	16#000005B8:
		F_EtherCAT_VendorIDtoString := 'Tarasheh System Pishro (tsPishro) Co., Ltd.';

	16#000005B9:
		F_EtherCAT_VendorIDtoString := 'CS-Lab s.c. Janusz Wawak, Andrzej Rogozynski, Szymon Paprocki';

	16#000005BA:
		F_EtherCAT_VendorIDtoString := 'Elitron IPM s.r.l.';

	16#000005BB:
		F_EtherCAT_VendorIDtoString := 'KORYO ELECTRONICS CO.,LTD.';

	16#000005BC:
		F_EtherCAT_VendorIDtoString := 'Shihlin Electric & Engineering Corporation';

	16#000005BD:
		F_EtherCAT_VendorIDtoString := 'Kookmin University, Graduate School of Automotive Engineering';

	16#000005BE:
		F_EtherCAT_VendorIDtoString := 'Techmation Co., Ltd.';

	16#000005BF:
		F_EtherCAT_VendorIDtoString := 'ZAPI S.p.A.';

	16#000005C0:
		F_EtherCAT_VendorIDtoString := 'Claus Pribbernow Mikrosystementwicklung eProcessorSolutions';

	16#000005C1:
		F_EtherCAT_VendorIDtoString := 'Pragati Automation Pvt. Ltd.';

	16#000005C2:
		F_EtherCAT_VendorIDtoString := 'Siemens Industry Software B.V.';

	16#000005C3:
		F_EtherCAT_VendorIDtoString := 'MicroNova AG';

	16#000005C4:
		F_EtherCAT_VendorIDtoString := 'XiAn Aerospace Precision Electromechanical Institute';

	16#000005C5:
		F_EtherCAT_VendorIDtoString := 'Dr. Mergenthaler GmbH & Co. KG';

	16#000005C6:
		F_EtherCAT_VendorIDtoString := 'China National Machinery Industry Corporation';

	16#000005C7:
		F_EtherCAT_VendorIDtoString := 'Berufliches Schulzentrum Hof, Staatliche Fachschule fur Technik';

	16#000005C8:
		F_EtherCAT_VendorIDtoString := 'NDR Co., Ltd';

	16#000005C9:
		F_EtherCAT_VendorIDtoString := '"NPK MSA" LLC';

	16#000005CA:
		F_EtherCAT_VendorIDtoString := 'Southeast University, School of Mechanical Engineering';

	16#000005CB:
		F_EtherCAT_VendorIDtoString := 'Shanghai Baosight Software Co., Ltd.';

	16#000005CC:
		F_EtherCAT_VendorIDtoString := 'Hakko Electronics Co., Ltd.';

	16#000005CD:
		F_EtherCAT_VendorIDtoString := 'GMK electronic design GmbH';

	16#000005CE:
		F_EtherCAT_VendorIDtoString := 'SIMTEC Elektronik GmbH';

	16#000005D0:
		F_EtherCAT_VendorIDtoString := 'TEConcept GmbH';

	16#000005D1:
		F_EtherCAT_VendorIDtoString := 'ESS Co., Ltd.';

	16#000005D3:
		F_EtherCAT_VendorIDtoString := 'MABI AG - Robotic';

	16#000005D4:
		F_EtherCAT_VendorIDtoString := 'OnRobot Hungary Kft';

	16#000005D5:
		F_EtherCAT_VendorIDtoString := 'TMEIC Corporation';

	16#000005D6:
		F_EtherCAT_VendorIDtoString := 'WITTENSTEIN ternary Co.,Ltd.';

	16#000005D7:
		F_EtherCAT_VendorIDtoString := 'Shanghai Friendess Electronic Technology Co., Ltd.';

	16#000005D8:
		F_EtherCAT_VendorIDtoString := 'Aversan Inc.';

	16#000005DA:
		F_EtherCAT_VendorIDtoString := 'Lorch Schweitechnik GmbH';

	16#000005D9:
		F_EtherCAT_VendorIDtoString := 'LOTES (GuangZhou) CO., LTD.';

	16#000005DB:
		F_EtherCAT_VendorIDtoString := 'Sungkyunkwan University, School of Mechanical Engineering';

	16#000005DC:
		F_EtherCAT_VendorIDtoString := 'Tsinghua University, Graduate School at Shenzhen';

	16#000005DD:
		F_EtherCAT_VendorIDtoString := 'Universidad de los Andes, Faculty of Engineering';

	16#000005DE:
		F_EtherCAT_VendorIDtoString := 'PFU LIMITED';

	16#000005DF:
		F_EtherCAT_VendorIDtoString := 'Slovak University of Technology in Bratislava, Faculty of Electrical Engineering and Information Technology';

	16#000005E0:
		F_EtherCAT_VendorIDtoString := 'Esomatec GmbH';

	16#000005E1:
		F_EtherCAT_VendorIDtoString := 'LS ELECTRIC Co., Ltd.';

	16#000005E2:
		F_EtherCAT_VendorIDtoString := 'StateCore B.V.';

	16#000005E3:
		F_EtherCAT_VendorIDtoString := 'KJ-Infinity Enterprises Inc.';

	16#000005E4:
		F_EtherCAT_VendorIDtoString := 'Center of Human-centered Interaction for Coexistence (CHIC)';

	16#000005E5:
		F_EtherCAT_VendorIDtoString := 'Littelfuse Selco A/S';

	16#000005E6:
		F_EtherCAT_VendorIDtoString := 'ITR GmbH Informationstechnologie Rauch';

	16#000005E8:
		F_EtherCAT_VendorIDtoString := 'University of Massachusetts at Amherst, Computer Science Department, Laboratory for Perceptual Robotics';

	16#000005E9:
		F_EtherCAT_VendorIDtoString := 'Pfeiffer Vacuum SAS';

	16#000005EA:
		F_EtherCAT_VendorIDtoString := 'AXOR INDUSTRIES s.n.c.';

	16#000005EB:
		F_EtherCAT_VendorIDtoString := 'QuadRep Electronics (Taiwan) Ltd.';

	16#000005EC:
		F_EtherCAT_VendorIDtoString := 'Herrmann Ultraschalltechnik GmbH & Co. KG';

	16#000005ED:
		F_EtherCAT_VendorIDtoString := 'Precizika Metrology, UAB';

	16#000005EE:
		F_EtherCAT_VendorIDtoString := 'Shanghai ReCAT Automation Control Technology Co., Ltd.';

	16#000005EF:
		F_EtherCAT_VendorIDtoString := 'U&R GmbH Hardware- und Systemdesign';

	16#000005F0:
		F_EtherCAT_VendorIDtoString := 'XiaMen MicroControl Technology Co., Ltd.';

	16#000005F1:
		F_EtherCAT_VendorIDtoString := 'The Oilgear Company';

	16#000005F2:
		F_EtherCAT_VendorIDtoString := 'MIE ELECTRONICS CO.,LTD. iSPC';

	16#000005F3:
		F_EtherCAT_VendorIDtoString := 'in-tech GmbH';

	16#000005F5:
		F_EtherCAT_VendorIDtoString := 'Starflight Electronics';

	16#000005F6:
		F_EtherCAT_VendorIDtoString := 'ZIEHL-ABEGG SE';

	16#000005F7:
		F_EtherCAT_VendorIDtoString := 'Ackermann Automation GmbH';

	16#000005F8:
		F_EtherCAT_VendorIDtoString := 'Helios Technologies, Inc.';

	16#000005F9:
		F_EtherCAT_VendorIDtoString := 'Italsensor s.r.l.';

	16#000005FA:
		F_EtherCAT_VendorIDtoString := 'Minebea Intec Aachen GmbH & Co. KG';

	16#000005FB:
		F_EtherCAT_VendorIDtoString := 'Evergrid Solutions & Systems';

	16#000005FC:
		F_EtherCAT_VendorIDtoString := 'Germanjet Company Limited';

	16#000005FD:
		F_EtherCAT_VendorIDtoString := 'Mapacode Inc.';

	16#000005FE:
		F_EtherCAT_VendorIDtoString := 'BIBA - Bremer Institut fur Produktion und Logistik GmbH';

	16#000005FF:
		F_EtherCAT_VendorIDtoString := 'The University of Texas at Austin';

	16#00000600:
		F_EtherCAT_VendorIDtoString := 'OKI Nextech Co.,Ltd.';

	16#00000601:
		F_EtherCAT_VendorIDtoString := 'Condalo GmbH';

	16#00000602:
		F_EtherCAT_VendorIDtoString := 'Brooks Instrument, LLC';

	16#00000603:
		F_EtherCAT_VendorIDtoString := 'FLORIDA INSTITUTE FOR HUMAN & MACHINE COGNITION';

	16#00000604:
		F_EtherCAT_VendorIDtoString := 'Leica Geosystems AG';

	16#00000605:
		F_EtherCAT_VendorIDtoString := 'Nabtesco Corporation';

	16#00000606:
		F_EtherCAT_VendorIDtoString := 'BP&M Representacoes e Consultoria LTDA';

	16#00000607:
		F_EtherCAT_VendorIDtoString := 'MICRO-EPSILON Optronic GmbH';

	16#00000608:
		F_EtherCAT_VendorIDtoString := 'Diamond Technologies, Inc.';

	16#0000060A:
		F_EtherCAT_VendorIDtoString := 'ESTUN AUTOMATION CO.,LTD';

	16#0000060B:
		F_EtherCAT_VendorIDtoString := 'IMS Messsysteme GmbH';

	16#0000060C:
		F_EtherCAT_VendorIDtoString := 'MG Co., Ltd.';

	16#0000060D:
		F_EtherCAT_VendorIDtoString := 'Ferrotec (USA) Corporation - Temescal Division';

	16#0000060E:
		F_EtherCAT_VendorIDtoString := 'SICK IVP AB';

	16#0000060F:
		F_EtherCAT_VendorIDtoString := 'Oregon State University, School of Mechanical, Industrial and Manufacturing Engineering';

	16#00000610:
		F_EtherCAT_VendorIDtoString := 'SINFONIA TECHNOLOGY CO., LTD.';

	16#00000611:
		F_EtherCAT_VendorIDtoString := 'Pfeiffer Vacuum GmbH';

	16#00000612:
		F_EtherCAT_VendorIDtoString := 'Froude Hofmann Limited';

	16#00000613:
		F_EtherCAT_VendorIDtoString := 'SABO Elektronik GmbH';

	16#00000615:
		F_EtherCAT_VendorIDtoString := 'Bystronic Laser AG';

	16#00000616:
		F_EtherCAT_VendorIDtoString := 'Shanghai Kinway Technologies, Inc.';

	16#00000617:
		F_EtherCAT_VendorIDtoString := 'Avnet K.K.';

	16#00000618:
		F_EtherCAT_VendorIDtoString := 'LumaSense Technologies GmbH';

	16#00000619:
		F_EtherCAT_VendorIDtoString := 'BBH Products GmbH';

	16#0000061A:
		F_EtherCAT_VendorIDtoString := 'Hecht Automatisierungs-Systeme GmbH';

	16#0000061B:
		F_EtherCAT_VendorIDtoString := 'Xelmo AB';

	16#0000061C:
		F_EtherCAT_VendorIDtoString := 'Carl Zeiss Industrielle Messtechnik GmbH';

	16#0000061D:
		F_EtherCAT_VendorIDtoString := 'University of Genova, Faculty of Engineering';

	16#0000061E:
		F_EtherCAT_VendorIDtoString := 'JOT Automation Oy';

	16#0000061F:
		F_EtherCAT_VendorIDtoString := 'Sankyo Seisakusho Co.';

	16#00000620:
		F_EtherCAT_VendorIDtoString := 'ATV-Elektronik Ges.m.b.H.';

	16#00000621:
		F_EtherCAT_VendorIDtoString := 'Panasonic Industry Co., Ltd.';

	16#00000622:
		F_EtherCAT_VendorIDtoString := 'ifm electronic gmbh';

	16#00000623:
		F_EtherCAT_VendorIDtoString := 'Fisher Technical Services Inc.';

	16#00000624:
		F_EtherCAT_VendorIDtoString := 'SCLE SFE';

	16#00000625:
		F_EtherCAT_VendorIDtoString := 'HIGEN RNM Co., Ltd.';

	16#00000626:
		F_EtherCAT_VendorIDtoString := 'Baumer hhs GmbH';

	16#00000627:
		F_EtherCAT_VendorIDtoString := 'Moog Inc.';

	16#00000628:
		F_EtherCAT_VendorIDtoString := 'XIOS Hogeschool Limburg, Department N-Technology';

	16#00000629:
		F_EtherCAT_VendorIDtoString := 'Azbil Corporation';

	16#0000062A:
		F_EtherCAT_VendorIDtoString := 'Delta Tau Data Systems, Inc.';

	16#0000062B:
		F_EtherCAT_VendorIDtoString := 'Heraeus Electro-Nite International N.V.';

	16#0000062C:
		F_EtherCAT_VendorIDtoString := 'ESW GmbH';

	16#0000062D:
		F_EtherCAT_VendorIDtoString := 'CG Drives & Automation AB';

	16#0000062E:
		F_EtherCAT_VendorIDtoString := 'ProCom GmbH';

	16#0000062F:
		F_EtherCAT_VendorIDtoString := 'GE Grid Solutions SAS';

	16#00000630:
		F_EtherCAT_VendorIDtoString := 'Robot Makers GmbH';

	16#00000631:
		F_EtherCAT_VendorIDtoString := 'Brooks Automation, Inc';

	16#00000632:
		F_EtherCAT_VendorIDtoString := 'Kuwana Metals, Ltd.';

	16#00000633:
		F_EtherCAT_VendorIDtoString := 'Interroll Automation GmbH';

	16#00000634:
		F_EtherCAT_VendorIDtoString := 'CKD Corporation';

	16#00000635:
		F_EtherCAT_VendorIDtoString := 'STIWA Automation GmbH';

	16#00000636:
		F_EtherCAT_VendorIDtoString := 'T.P.A. S.p.A';

	16#00000637:
		F_EtherCAT_VendorIDtoString := 'Guodian Nanjing Automation Co., Ltd.';

	16#00000638:
		F_EtherCAT_VendorIDtoString := 'Prosoft-Systems Ltd.';

	16#00000639:
		F_EtherCAT_VendorIDtoString := 'Polytype SA';

	16#0000063A:
		F_EtherCAT_VendorIDtoString := 'SENSODRIVE GmbH';

	16#0000063B:
		F_EtherCAT_VendorIDtoString := 'Delta Computer Systems, Inc.';

	16#0000063C:
		F_EtherCAT_VendorIDtoString := 'Friedrich Lutze GmbH';

	16#0000063D:
		F_EtherCAT_VendorIDtoString := 'Compressor Controls Corporation';

	16#0000063E:
		F_EtherCAT_VendorIDtoString := 'Diamond Light Source Limited';

	16#0000063F:
		F_EtherCAT_VendorIDtoString := 'Beckman Coulter, Inc.';

	16#00000640:
		F_EtherCAT_VendorIDtoString := 'Allied Motion Technologies, Inc.';

	16#00000641:
		F_EtherCAT_VendorIDtoString := 'Nor-Cal Products, Inc.';

	16#00000642:
		F_EtherCAT_VendorIDtoString := 'AUTOMATA GmbH & Co. KG';

	16#00000643:
		F_EtherCAT_VendorIDtoString := 'Fraunhofer-Institut fur Werkstoff- und Strahltechnik IWS';

	16#00000644:
		F_EtherCAT_VendorIDtoString := 'INFICON AG';

	16#00000645:
		F_EtherCAT_VendorIDtoString := 'Hexagon Metrology GmbH';

	16#00000646:
		F_EtherCAT_VendorIDtoString := 'Shimadzu Corporation';

	16#00000647:
		F_EtherCAT_VendorIDtoString := 'Dasa Control Systems AB';

	16#00000648:
		F_EtherCAT_VendorIDtoString := 'SHOEI Electric Co.,Ltd.';

	16#00000649:
		F_EtherCAT_VendorIDtoString := 'Progressio, LLC';

	16#0000064A:
		F_EtherCAT_VendorIDtoString := 'MACCON GmbH & Co. KG';

	16#0000064B:
		F_EtherCAT_VendorIDtoString := 'Moog Ireland, Ltd.';

	16#0000064C:
		F_EtherCAT_VendorIDtoString := 'ESPERA-WERKE GMBH';

	16#0000064D:
		F_EtherCAT_VendorIDtoString := 'Automation W+R GmbH';

	16#0000064E:
		F_EtherCAT_VendorIDtoString := 'Oceaneering Space Systems';

	16#0000064F:
		F_EtherCAT_VendorIDtoString := 'EOStech S.r.l.';

	16#00000650:
		F_EtherCAT_VendorIDtoString := 'Lycee Jean-Baptiste de Baudre';

	16#00000651:
		F_EtherCAT_VendorIDtoString := 'University of Banja Luka';

	16#00000652:
		F_EtherCAT_VendorIDtoString := 'Eding CNC';

	16#00000653:
		F_EtherCAT_VendorIDtoString := 'Zuhlke Engineering AG';

	16#00000654:
		F_EtherCAT_VendorIDtoString := 'Addiva Consulting AB';

	16#00000655:
		F_EtherCAT_VendorIDtoString := 'Pteris Global Limited';

	16#00000656:
		F_EtherCAT_VendorIDtoString := 'Chaos Technology';

	16#00000657:
		F_EtherCAT_VendorIDtoString := 'Tokyo Institute of Technology, Hirose Fukushima Lab.';

	16#00000658:
		F_EtherCAT_VendorIDtoString := 'Seichter GmbH';

	16#00000659:
		F_EtherCAT_VendorIDtoString := 'Motion Control Systems, Inc.';

	16#0000065A:
		F_EtherCAT_VendorIDtoString := 'Moog B.V.';

	16#0000065B:
		F_EtherCAT_VendorIDtoString := 'Kinlo Technology & System (Shenzhen) Co.,Ltd.';

	16#0000065C:
		F_EtherCAT_VendorIDtoString := 'CellSystems, LLC';

	16#0000065D:
		F_EtherCAT_VendorIDtoString := 'Shinano Kenshi Co., Ltd.';

	16#0000065E:
		F_EtherCAT_VendorIDtoString := 'MICRO-EPSILON MESSTECHNIK GmbH & Co. KG';

	16#0000065F:
		F_EtherCAT_VendorIDtoString := 'Viable Bytes, Inc.';

	16#00000660:
		F_EtherCAT_VendorIDtoString := 'Kontron Europe GmbH';

	16#00000661:
		F_EtherCAT_VendorIDtoString := 'IKERLAN, S. Coop.';

	16#00000662:
		F_EtherCAT_VendorIDtoString := 'hmk Daten-System-Technik GmbH';

	16#00000664:
		F_EtherCAT_VendorIDtoString := 'Istituto Italiano di Tecnologia (IIT)';

	16#00000663:
		F_EtherCAT_VendorIDtoString := 'Qingdao INCMAN Robot Co., Ltd.';

	16#00000665:
		F_EtherCAT_VendorIDtoString := 'Kashiyama Industries, Ltd.';

	16#00000666:
		F_EtherCAT_VendorIDtoString := 'TG Drives s.r.o.';

	16#00000667:
		F_EtherCAT_VendorIDtoString := 'Watlow Electric Manufacturing Company';

	16#00000668:
		F_EtherCAT_VendorIDtoString := 'synertronixx GmbH';

	16#00000669:
		F_EtherCAT_VendorIDtoString := 'batalpha Bobach GmbH';

	16#0000066A:
		F_EtherCAT_VendorIDtoString := 'Edwards Limited';

	16#0000066B:
		F_EtherCAT_VendorIDtoString := 'ENGEL AUSTRIA GmbH';

	16#0000066C:
		F_EtherCAT_VendorIDtoString := 'Fujikin Incorporated';

	16#0000066D:
		F_EtherCAT_VendorIDtoString := 'COMET Technologies USA, Inc.';

	16#0000066E:
		F_EtherCAT_VendorIDtoString := 'Schleuniger AG';

	16#0000066F:
		F_EtherCAT_VendorIDtoString := 'Panasonic Industry Co., Ltd.';

	16#00000670:
		F_EtherCAT_VendorIDtoString := 'TangShan Kaiyuan Welding Automation Technology Institute Co., Ltd.';

	16#00000671:
		F_EtherCAT_VendorIDtoString := 'Solectrix GmbH';

	16#00000672:
		F_EtherCAT_VendorIDtoString := 'St. Cloud State University, Electrical and Computer Engineering Department';

	16#00000673:
		F_EtherCAT_VendorIDtoString := 'JLG AUTOMATION BVBA';

	16#00000674:
		F_EtherCAT_VendorIDtoString := 'Burckhardt Compression AG';

	16#00000675:
		F_EtherCAT_VendorIDtoString := 'Rong Shun Xuan Corp.';

	16#00000676:
		F_EtherCAT_VendorIDtoString := 'Balluff STM GmbH';

	16#00000677:
		F_EtherCAT_VendorIDtoString := 'Endress+Hauser Flowtec AG';

	16#00000678:
		F_EtherCAT_VendorIDtoString := 'Motor Power Company S.r.l.';

	16#0000067A:
		F_EtherCAT_VendorIDtoString := 'EBI Electric Inc.';

	16#0000067B:
		F_EtherCAT_VendorIDtoString := 'Hochschule Luzern, Technik & Architektur';

	16#0000067C:
		F_EtherCAT_VendorIDtoString := 'GE Global Research';

	16#0000067D:
		F_EtherCAT_VendorIDtoString := 'Katholieke Universiteit Leuven, Department of Mechanical Engineering';

	16#0000067E:
		F_EtherCAT_VendorIDtoString := 'centrotherm international AG';

	16#0000067F:
		F_EtherCAT_VendorIDtoString := 'Bundesamt fur Wehrtechnik und Beschaffung, Wehrtechnische Dienststelle fur Informationstechnologie und Elektronik (WTD 81)';

	16#00000680:
		F_EtherCAT_VendorIDtoString := 'DAIHEN Corporation';

	16#00000681:
		F_EtherCAT_VendorIDtoString := 'HCL Technologies Ltd.';

	16#00000682:
		F_EtherCAT_VendorIDtoString := '3T B.V.';

	16#00000683:
		F_EtherCAT_VendorIDtoString := 'Eindhoven University of Technology';

	16#00000684:
		F_EtherCAT_VendorIDtoString := 'INNOVENT e.V.';

	16#00000685:
		F_EtherCAT_VendorIDtoString := 'Surrey Satellite Technology Limited';

	16#00000686:
		F_EtherCAT_VendorIDtoString := 'AMETEK Programmable Power, Inc.';

	16#00000687:
		F_EtherCAT_VendorIDtoString := 'engleder embedded';

	16#00000688:
		F_EtherCAT_VendorIDtoString := 'Pusan National University';

	16#00000689:
		F_EtherCAT_VendorIDtoString := 'ETH Zurich, Institute of Robotics and Intelligent Systems (IRIS)';

	16#0000068A:
		F_EtherCAT_VendorIDtoString := 'Expleo Germany GmbH';

	16#0000068B:
		F_EtherCAT_VendorIDtoString := 'HORIBA, Ltd.';

	16#0000068C:
		F_EtherCAT_VendorIDtoString := 'Changwon National University, College of Engineering, Department of Electrical Engineering';

	16#0000068D:
		F_EtherCAT_VendorIDtoString := 'Penko Engineering B.V.';

	16#0000068E:
		F_EtherCAT_VendorIDtoString := 'Fujitsu Semiconductor Europe GmbH';

	16#00000690:
		F_EtherCAT_VendorIDtoString := 'Mirle Automation Corporation';

	16#00000691:
		F_EtherCAT_VendorIDtoString := 'FANUC CORPORATION';

	16#00000692:
		F_EtherCAT_VendorIDtoString := 'KSE GmbH';

	16#00000693:
		F_EtherCAT_VendorIDtoString := 'EUCHNER GmbH + Co. KG';

	16#00000694:
		F_EtherCAT_VendorIDtoString := 'benjamin GmbH';

	16#00000695:
		F_EtherCAT_VendorIDtoString := 'Hans Laser Technology Co.,Ltd.';

	16#00000696:
		F_EtherCAT_VendorIDtoString := 'Guangdong University of Technology, Faculty of Automation';

	16#00000699:
		F_EtherCAT_VendorIDtoString := 'Instituto Federal de Santa Catarina';

	16#0000069A:
		F_EtherCAT_VendorIDtoString := 'InstruTech Inc.';

	16#0000069B:
		F_EtherCAT_VendorIDtoString := 'KTL Corporation';

	16#0000069C:
		F_EtherCAT_VendorIDtoString := 'Hochschule Pforzheim, Fakultat fur Technik';

	16#0000069D:
		F_EtherCAT_VendorIDtoString := 'EWM HIGHTEC WELDING GmbH';

	16#0000069E:
		F_EtherCAT_VendorIDtoString := 'Jilin Yongda Group Company Ltd.';

	16#0000069F:
		F_EtherCAT_VendorIDtoString := 'Arrow Central Europe GmbH';

	16#000006A0:
		F_EtherCAT_VendorIDtoString := 'Phoseon Technology';

	16#000006A1:
		F_EtherCAT_VendorIDtoString := 'item Industrietechnik GmbH';

	16#000006A2:
		F_EtherCAT_VendorIDtoString := 'Shanghai Inno-drive Electric Co., Ltd.';

	16#000006A3:
		F_EtherCAT_VendorIDtoString := 'Wuhan University of Technology, School of Automation';

	16#000006A4:
		F_EtherCAT_VendorIDtoString := 'Advanet Inc.';

	16#000006A5:
		F_EtherCAT_VendorIDtoString := 'Wandercraft SAS';

	16#000006A6:
		F_EtherCAT_VendorIDtoString := 'Changzhou Xiangyun Monitoring Software Co., Ltd.';

	16#000006A7:
		F_EtherCAT_VendorIDtoString := 'SANTEST CO., LTD.';

	16#000006A8:
		F_EtherCAT_VendorIDtoString := 'EnTeSys GmbH';

	16#000006A9:
		F_EtherCAT_VendorIDtoString := 'LOT Vacuum Co., Ltd.';

	16#000006AA:
		F_EtherCAT_VendorIDtoString := 'ASM America Inc.';

	16#000006AB:
		F_EtherCAT_VendorIDtoString := 'Taiwan Pulse Motion Co. Ltd.';

	16#000006AC:
		F_EtherCAT_VendorIDtoString := 'CNi Informatica S.r.l.';

	16#000006AD:
		F_EtherCAT_VendorIDtoString := 'enfas GmbH';

	16#000006AE:
		F_EtherCAT_VendorIDtoString := 'Shenzhen Megmeet Drive Technology Co., Ltd.';

	16#000006AF:
		F_EtherCAT_VendorIDtoString := 'Danish Aerospace Company';

	16#000006B0:
		F_EtherCAT_VendorIDtoString := 'Panasonic Production Engineering Co., Ltd.';

	16#000006B1:
		F_EtherCAT_VendorIDtoString := 'ARADEX AG';

	16#000006B2:
		F_EtherCAT_VendorIDtoString := 'TOYOGIKEN CO.,LTD.';

	16#000006B3:
		F_EtherCAT_VendorIDtoString := 'ZAO Trascon Technology';

	16#000006B4:
		F_EtherCAT_VendorIDtoString := 'AREM PRO, s.r.o.';

	16#000006B5:
		F_EtherCAT_VendorIDtoString := 'Googol Technology Co. Ltd.';

	16#000006B6:
		F_EtherCAT_VendorIDtoString := 'Vecna Technologies, Inc.';

	16#000006B7:
		F_EtherCAT_VendorIDtoString := 'Technische Universitat Dresden, Fakultat Elektrotechnik und Informationstechnik';

	16#000006B8:
		F_EtherCAT_VendorIDtoString := 'Axxon Computer Corporation';

	16#000006B9:
		F_EtherCAT_VendorIDtoString := 'Beijing Motrotech Technology Co., Ltd.';

	16#000006BA:
		F_EtherCAT_VendorIDtoString := 'Wohner GmbH & Co. KG';

	16#000006BB:
		F_EtherCAT_VendorIDtoString := 'Hangzhou Tongling Automation Co., Ltd.';

	16#000006BC:
		F_EtherCAT_VendorIDtoString := 'Audix Corporation';

	16#000006BD:
		F_EtherCAT_VendorIDtoString := 'Technische Universitat Wien, Fakultat fur Elektrotechnik und Informationstechnik';

	16#000006BE:
		F_EtherCAT_VendorIDtoString := 'AREVA NP';

	16#000006BF:
		F_EtherCAT_VendorIDtoString := 'TAURUS instruments GmbH';

	16#000006C0:
		F_EtherCAT_VendorIDtoString := 'Aveox Inc.';

	16#000006C1:
		F_EtherCAT_VendorIDtoString := 'ASML Netherlands B.V.';

	16#000006C2:
		F_EtherCAT_VendorIDtoString := 'HaslerRail AG';

	16#000006C3:
		F_EtherCAT_VendorIDtoString := 'Intek Technology Co., Ltd.';

	16#000006C4:
		F_EtherCAT_VendorIDtoString := 'National Computer System Engineering Research Institute of China';

	16#000006C5:
		F_EtherCAT_VendorIDtoString := 'Crouzet Automatismes';

	16#000006C7:
		F_EtherCAT_VendorIDtoString := 'Joshua 1 Systems Inc.';

	16#000006C8:
		F_EtherCAT_VendorIDtoString := 'Artech Electronics Co., Ltd.';

	16#000006CA:
		F_EtherCAT_VendorIDtoString := 'FUJI MACHINERY CO.,LTD.';

	16#000006CB:
		F_EtherCAT_VendorIDtoString := 'FoShan Logen Robotics Co., Ltd.';

	16#000006CC:
		F_EtherCAT_VendorIDtoString := 'DVDB-electronics bvba';

	16#000006CD:
		F_EtherCAT_VendorIDtoString := 'Tool Express-Service Schraubertechnik GmbH';

	16#000006CE:
		F_EtherCAT_VendorIDtoString := 'King Giants Precision Industry Co., Ltd.';

	16#000006CF:
		F_EtherCAT_VendorIDtoString := 'PANAX SYSTEM Co., Ltd.';

	16#000006D0:
		F_EtherCAT_VendorIDtoString := 'Hitachi Europe GmbH';

	16#000006D1:
		F_EtherCAT_VendorIDtoString := 'ZDAUTO AZDAUTO Automation Technology Co., Ltd. utomation Technology Co., Ltd.';

	16#000006D2:
		F_EtherCAT_VendorIDtoString := 'Temis S.r.l.';

	16#000006D3:
		F_EtherCAT_VendorIDtoString := 'DAIKIN INDUSTRIES, LTD., Oil Hydraulics Division';

	16#000006D4:
		F_EtherCAT_VendorIDtoString := 'Avalue Technology Inc.';

	16#000006D5:
		F_EtherCAT_VendorIDtoString := 'LDZ Technology Co., Ltd.';

	16#000006D6:
		F_EtherCAT_VendorIDtoString := 'Eletech S.r.l.';

	16#000006D9:
		F_EtherCAT_VendorIDtoString := 'Portwell, Inc.';

	16#000006DA:
		F_EtherCAT_VendorIDtoString := 'Shenzhen Sine Electric Co., Ltd';

	16#000006DB:
		F_EtherCAT_VendorIDtoString := 'HIMA Paul Hildebrandt GmbH';

	16#000006DC:
		F_EtherCAT_VendorIDtoString := 'Covidien LP';

	16#000006DD:
		F_EtherCAT_VendorIDtoString := 'Weintek IIoT HK Ltd., Taiwan Branch';

	16#000006DE:
		F_EtherCAT_VendorIDtoString := 'MITWELL Inc.';

	16#000006DF:
		F_EtherCAT_VendorIDtoString := 'DORNA Technology Co., Ltd.';

	16#000006E0:
		F_EtherCAT_VendorIDtoString := 'A M Consulting';

	16#000006E1:
		F_EtherCAT_VendorIDtoString := 'GENESI ELETTRONICA Srl';

	16#000006E2:
		F_EtherCAT_VendorIDtoString := 'Molex Canada Limited';

	16#000006E3:
		F_EtherCAT_VendorIDtoString := 'Vanguard Systems Inc.';

	16#000006E4:
		F_EtherCAT_VendorIDtoString := 'Shenzhen UniMAT Automation Technology Co., Ltd.';

	16#000006E5:
		F_EtherCAT_VendorIDtoString := 'ifatos GmbH & Co. KG';

	16#000006E6:
		F_EtherCAT_VendorIDtoString := 'Ingenieria UNO S.L';

	16#000006E7:
		F_EtherCAT_VendorIDtoString := 'Daekhon Corporation';

	16#000006EA:
		F_EtherCAT_VendorIDtoString := 'Marubeni Information Systems Co., Ltd.';

	16#000006EB:
		F_EtherCAT_VendorIDtoString := 'YDK Co., Ltd.';

	16#000006EC:
		F_EtherCAT_VendorIDtoString := 'E-T-A Elektrotechnische Apparate GmbH';

	16#000006EE:
		F_EtherCAT_VendorIDtoString := 'Justech Precision Industry Co., Ltd.';

	16#000006F0:
		F_EtherCAT_VendorIDtoString := 'VOLLMER WERKE Maschinenfabrik GmbH';

	16#000006F1:
		F_EtherCAT_VendorIDtoString := 'Technische Hochschule Nurnberg Georg Simon Ohm';

	16#000006F2:
		F_EtherCAT_VendorIDtoString := 'Gene Automation Technology Ltd.';

	16#000006F3:
		F_EtherCAT_VendorIDtoString := 'Weihai Zheng Qi Mechatronics Technology Ltd.';

	16#000006F5:
		F_EtherCAT_VendorIDtoString := 'Gopher Inc.';

	16#000006F6:
		F_EtherCAT_VendorIDtoString := 'IntervalZero, Inc.';

	16#000006F7:
		F_EtherCAT_VendorIDtoString := 'AXONIM LLC';

	16#000006F8:
		F_EtherCAT_VendorIDtoString := 'University of Seoul, College of Engineering, Department of Mechanical and Information Engineering';

	16#000006F9:
		F_EtherCAT_VendorIDtoString := 'Professional Computer Technology Limited';

	16#000006FA:
		F_EtherCAT_VendorIDtoString := 'Ninna Solutions Co,.Ltd';

	16#000006FC:
		F_EtherCAT_VendorIDtoString := 'Shenyang CASNC Technology Co., Ltd.';

	16#000006FD:
		F_EtherCAT_VendorIDtoString := 'IWAKI CO., LTD.';

	16#000006FE:
		F_EtherCAT_VendorIDtoString := 'TRP Engineering College, Department of Electronics & Communication Engineering (ECE)';

	16#000006FF:
		F_EtherCAT_VendorIDtoString := 'EPI elettronica s.a.s.';

	16#00000700:
		F_EtherCAT_VendorIDtoString := 'Institut de RadioAstronomie Millimetrique';

	16#00000701:
		F_EtherCAT_VendorIDtoString := 'Technische Universitat Graz, Fakultat fur Maschinenbau und Wirtschaftswissenschaften';

	16#00000702:
		F_EtherCAT_VendorIDtoString := 'pro-beam AG & Co. KGaA';

	16#00000703:
		F_EtherCAT_VendorIDtoString := 'Servotechnica ZAO';

	16#00000704:
		F_EtherCAT_VendorIDtoString := 'Hanwha Precision Machinery CO., LTD.';

	16#00000705:
		F_EtherCAT_VendorIDtoString := 'G&S Intelligent Technology Co., Ltd.';

	16#00000706:
		F_EtherCAT_VendorIDtoString := 'Schaeffler Engineering';

	16#00000707:
		F_EtherCAT_VendorIDtoString := 'University of the Basque Country, Faculty of Engineering of Bilbao, Department of Electronics and Telecommunications';

	16#00000708:
		F_EtherCAT_VendorIDtoString := 'ARGES GmbH';

	16#00000709:
		F_EtherCAT_VendorIDtoString := 'Control Chief Corporation';

	16#0000070A:
		F_EtherCAT_VendorIDtoString := 'konplan systemhaus ag';

	16#0000070B:
		F_EtherCAT_VendorIDtoString := 'embeX GmbH';

	16#0000070C:
		F_EtherCAT_VendorIDtoString := 'COSMOTECHS Co., Ltd';

	16#0000070D:
		F_EtherCAT_VendorIDtoString := 'Dynamic Systems Inc.';

	16#0000070E:
		F_EtherCAT_VendorIDtoString := 'SEMIKRON Elektronik GmbH & Co. KG';

	16#0000070F:
		F_EtherCAT_VendorIDtoString := 'Wuxi Ivoyage Control Technology CO.,LTD';

	16#00000710:
		F_EtherCAT_VendorIDtoString := 'CAF Signalling S.L.';

	16#00000711:
		F_EtherCAT_VendorIDtoString := 'SMART Electronic Development GmbH';

	16#00000712:
		F_EtherCAT_VendorIDtoString := 'Yokogawa Electric Corporation';

	16#00000713:
		F_EtherCAT_VendorIDtoString := 'Norwegian University of Science and Technoloogy, 
            Faculty of Information Technology, Mathematics and Electrical Engineering';

	16#00000714:
		F_EtherCAT_VendorIDtoString := 'Robostar Co., Ltd';

	16#00000715:
		F_EtherCAT_VendorIDtoString := 'TRUMPF Werkzeugmaschinen SE + Co. KG';

	16#00000716:
		F_EtherCAT_VendorIDtoString := 'High Performance Motion System Development Co., Ltd.';

	16#00000717:
		F_EtherCAT_VendorIDtoString := 'Kozaka Electronic Design Inc.';

	16#00000718:
		F_EtherCAT_VendorIDtoString := 'Aeronautical Systems Engineering Inc.';

	16#00000719:
		F_EtherCAT_VendorIDtoString := 'Agile Planet, Inc.';

	16#0000071A:
		F_EtherCAT_VendorIDtoString := 'Hon Hai Precision Industry Co., Ltd.';

	16#0000071B:
		F_EtherCAT_VendorIDtoString := 'Systeme + Steuerungen GmbH';

	16#0000071C:
		F_EtherCAT_VendorIDtoString := 'Huron Net Works, Inc.';

	16#0000071D:
		F_EtherCAT_VendorIDtoString := 'University of Applied Sciences of Southern Switzerland, Department of Innovative Technologies (DTI)';

	16#0000071E:
		F_EtherCAT_VendorIDtoString := 'MAKO Surgical Corp.';

	16#0000071F:
		F_EtherCAT_VendorIDtoString := 'Rainer Thomas Messtechnik GmbH';

	16#00000720:
		F_EtherCAT_VendorIDtoString := 'ELTEK spol. s r.o.';

	16#00000721:
		F_EtherCAT_VendorIDtoString := 'Vecow Co., Ltd.';

	16#00000722:
		F_EtherCAT_VendorIDtoString := 'M&P Motion Control and Power Electronics GmbH';

	16#00000723:
		F_EtherCAT_VendorIDtoString := 'Leybold GmbH';

	16#00000725:
		F_EtherCAT_VendorIDtoString := 'Panasonic Industrial Devices Sales Company of America';

	16#00000726:
		F_EtherCAT_VendorIDtoString := 'Eilersen Electric Digital Systems A/S';

	16#00000727:
		F_EtherCAT_VendorIDtoString := 'Inter Factory Partners Co., LTD.';

	16#00000728:
		F_EtherCAT_VendorIDtoString := 'Power Instrument Co., Ltd.';

	16#00000729:
		F_EtherCAT_VendorIDtoString := 'Cosworth Group Holdings Ltd';

	16#0000072A:
		F_EtherCAT_VendorIDtoString := 'South China University of Technology, School of Mechanical & Automotive Engineering';

	16#0000072B:
		F_EtherCAT_VendorIDtoString := 'WARWICK INSTRUMENTS LTD.';

	16#0000072C:
		F_EtherCAT_VendorIDtoString := 'Shenzhen INVT Electric Co., Ltd.';

	16#0000072D:
		F_EtherCAT_VendorIDtoString := 'WIEDEG Elektronik GmbH';

	16#0000072E:
		F_EtherCAT_VendorIDtoString := 'NKE corporation';

	16#0000072F:
		F_EtherCAT_VendorIDtoString := 'Universidad Politecnica de Madrid';

	16#00000730:
		F_EtherCAT_VendorIDtoString := 'Bot & Dolly';

	16#00000731:
		F_EtherCAT_VendorIDtoString := 'RECIF Technologies';

	16#00000732:
		F_EtherCAT_VendorIDtoString := 'ATI Industrial Automation';

	16#00000733:
		F_EtherCAT_VendorIDtoString := 'ADVANTEST CORPORATION';

	16#00000734:
		F_EtherCAT_VendorIDtoString := 'MULTIVAC Sepp Haggenmuller SE & Co. KG';

	16#00000735:
		F_EtherCAT_VendorIDtoString := 'ROLAND ELECTRONIC GmbH';

	16#00000736:
		F_EtherCAT_VendorIDtoString := 'CONTEC Co., Ltd.';

	16#00000737:
		F_EtherCAT_VendorIDtoString := 'Alizem Inc.';

	16#00000738:
		F_EtherCAT_VendorIDtoString := 'Chyng Hong Electronic Co., Ltd.';

	16#00000739:
		F_EtherCAT_VendorIDtoString := 'Yaskawa America Inc.';

	16#0000073A:
		F_EtherCAT_VendorIDtoString := 'Georg Schlegel GmbH & Co. KG';

	16#0000073B:
		F_EtherCAT_VendorIDtoString := 'Faraday Technology Corporation';

	16#0000073C:
		F_EtherCAT_VendorIDtoString := 'SIPRO S.r.l.';

	16#0000073D:
		F_EtherCAT_VendorIDtoString := 'University of Twente, Faculty of Engineering Technology (CTW)';

	16#0000073E:
		F_EtherCAT_VendorIDtoString := 'Aalborg University';

	16#0000073F:
		F_EtherCAT_VendorIDtoString := 'S-SYS bvba';

	16#00000740:
		F_EtherCAT_VendorIDtoString := 'Ningbo Mingpu Automation Technology Co.';

	16#00000741:
		F_EtherCAT_VendorIDtoString := 'elrest Automationssysteme GmbH';

	16#00000742:
		F_EtherCAT_VendorIDtoString := 'Kyosan Electric Manufacturing Co., Ltd.';

	16#00000743:
		F_EtherCAT_VendorIDtoString := 'Custom Machines';

	16#00000744:
		F_EtherCAT_VendorIDtoString := 'KFM Regelungstechnik GmbH';

	16#00000745:
		F_EtherCAT_VendorIDtoString := 'ISHIDA CO., LTD.';

	16#00000746:
		F_EtherCAT_VendorIDtoString := 'Beijing University of Technology';

	16#00000747:
		F_EtherCAT_VendorIDtoString := 'GENTEC TECHNOLOGIES CO., LTD.';

	16#00000748:
		F_EtherCAT_VendorIDtoString := 'Tsino-dynatron Electrical Technology Beijing Co., Ltd.';

	16#00000749:
		F_EtherCAT_VendorIDtoString := 'PENTA TRADING Spol. S.r.o.';

	16#0000074A:
		F_EtherCAT_VendorIDtoString := 'University of Electronic Science and Technology of China, School of Optoelectronic Information';

	16#0000074B:
		F_EtherCAT_VendorIDtoString := 'Altus Sistemas de Informatica S/A';

	16#0000074C:
		F_EtherCAT_VendorIDtoString := 'Sanming University, Sanming Mechanical CAD Engineering Research Center';

	16#0000074E:
		F_EtherCAT_VendorIDtoString := 'JENOPTIK Industrial Metrology Germany GmbH';

	16#0000074F:
		F_EtherCAT_VendorIDtoString := 'Beijing KND CNC Technique Co., Ltd.';

	16#00000750:
		F_EtherCAT_VendorIDtoString := 'JW Shannon Engineers';

	16#00000751:
		F_EtherCAT_VendorIDtoString := 'A2V Mecatronique SAS';

	16#00000752:
		F_EtherCAT_VendorIDtoString := 'NEXCOM International Co., Ltd.';

	16#00000753:
		F_EtherCAT_VendorIDtoString := 'Jiangyin Huafeng Printing Machinery Co., Ltd.';

	16#00000754:
		F_EtherCAT_VendorIDtoString := 'Lectra SA';

	16#00000755:
		F_EtherCAT_VendorIDtoString := 'Beijer Electronics Products AB';

	16#00000756:
		F_EtherCAT_VendorIDtoString := 'C J Hartman Elektronik AB';

	16#00000757:
		F_EtherCAT_VendorIDtoString := 'Hurco Automation Ltd.';

	16#00000759:
		F_EtherCAT_VendorIDtoString := 'Autonics Corporation';

	16#0000075A:
		F_EtherCAT_VendorIDtoString := 'Brom Mechatronica B.V.';

	16#0000075B:
		F_EtherCAT_VendorIDtoString := 'Vrije Universiteit Brussel, Faculty of Engineering';

	16#0000075C:
		F_EtherCAT_VendorIDtoString := 'Alluris GmbH & Co. KG';

	16#0000075D:
		F_EtherCAT_VendorIDtoString := 'Hochschule Offenburg, Fakultat Elektrotechnik und Informationstechnik';

	16#0000075E:
		F_EtherCAT_VendorIDtoString := 'Instron - Division of ITW Ltd.';

	16#0000075F:
		F_EtherCAT_VendorIDtoString := 'Heidolph Elektro GmbH & Co. KG';

	16#00000760:
		F_EtherCAT_VendorIDtoString := 'GE Transportation';

	16#00000761:
		F_EtherCAT_VendorIDtoString := 'MAX GmbH';

	16#00000762:
		F_EtherCAT_VendorIDtoString := 'Durst Phototechnik Digital Technology GmbH';

	16#00000763:
		F_EtherCAT_VendorIDtoString := 'Omsk State Technical University, Department of „Electricity industry“';

	16#00000764:
		F_EtherCAT_VendorIDtoString := 'Embedded-Bonjour GmbH';

	16#00000765:
		F_EtherCAT_VendorIDtoString := 'Mettler-Toledo Garvens GmbH';

	16#00000766:
		F_EtherCAT_VendorIDtoString := 'Renesas Electronics Corporation';

	16#00000767:
		F_EtherCAT_VendorIDtoString := 'Conductix-Wampfler Automation GmbH';

	16#00000768:
		F_EtherCAT_VendorIDtoString := 'EURA DRIVES ELECTRIC CO. LTD';

	16#00000769:
		F_EtherCAT_VendorIDtoString := 'EUTRON S.p.A.';

	16#0000076A:
		F_EtherCAT_VendorIDtoString := 'FLANDERS Inc.';

	16#0000076B:
		F_EtherCAT_VendorIDtoString := 'Digital Dynamics, Inc.';

	16#0000076C:
		F_EtherCAT_VendorIDtoString := 'GE Medical Systems Europe';

	16#0000076D:
		F_EtherCAT_VendorIDtoString := 'Physik Instrumente (PI) SE & Co. KG';

	16#0000076E:
		F_EtherCAT_VendorIDtoString := 'Hypertherm Inc.';

	16#0000076F:
		F_EtherCAT_VendorIDtoString := 'HRID d.o.o.';

	16#00000770:
		F_EtherCAT_VendorIDtoString := 'Aotai Electric Co., LTD';

	16#00000771:
		F_EtherCAT_VendorIDtoString := 'Control Concepts Inc.';

	16#00000772:
		F_EtherCAT_VendorIDtoString := 'JoveTech Co., Ltd.';

	16#00000773:
		F_EtherCAT_VendorIDtoString := 'POHANG UNIVERSITY OF SCIENCE AND TECHNOLOGY, Department of Electrical Engineering';

	16#00000774:
		F_EtherCAT_VendorIDtoString := 'CycloMedia Technology B.V.';

	16#00000775:
		F_EtherCAT_VendorIDtoString := 'SUN-TECTRO LTD.';

	16#00000776:
		F_EtherCAT_VendorIDtoString := 'Shanghai Jiao Tong University, School of Electronic Information and Electrical Engineering';

	16#00000777:
		F_EtherCAT_VendorIDtoString := 'koenig-pa GmbH';

	16#00000778:
		F_EtherCAT_VendorIDtoString := 'Anton Paar TriTec SA';

	16#00000779:
		F_EtherCAT_VendorIDtoString := 'V TEX Corporation';

	16#0000077A:
		F_EtherCAT_VendorIDtoString := 'Edge Technologies';

	16#0000077B:
		F_EtherCAT_VendorIDtoString := 'EBARA CORPORATION';

	16#0000077C:
		F_EtherCAT_VendorIDtoString := 'University at Buffalo';

	16#0000077D:
		F_EtherCAT_VendorIDtoString := 'Aurotek Corporation';

	16#0000077E:
		F_EtherCAT_VendorIDtoString := 'Blubit d.o.o.';

	16#0000077F:
		F_EtherCAT_VendorIDtoString := 'Toplens Hangzhou, Inc.';

	16#00000780:
		F_EtherCAT_VendorIDtoString := 'National Chung Cheng University';

	16#00000781:
		F_EtherCAT_VendorIDtoString := 'Hexagon Technology Center GmbH';

	16#00000782:
		F_EtherCAT_VendorIDtoString := 'Graph-Tech AG';

	16#00000783:
		F_EtherCAT_VendorIDtoString := 'Lanthan GmbH & Co. KG';

	16#00000784:
		F_EtherCAT_VendorIDtoString := 'Nucleus GmbH';

	16#00000785:
		F_EtherCAT_VendorIDtoString := 'BBULL Technology GmbH';

	16#00000786:
		F_EtherCAT_VendorIDtoString := 'Universitat Wien, Fakultat fur Physik, Isotopenforschung';

	16#00000787:
		F_EtherCAT_VendorIDtoString := 'inno-spec GmbH';

	16#00000788:
		F_EtherCAT_VendorIDtoString := 'ThyssenKrupp Presta AG';

	16#0000078A:
		F_EtherCAT_VendorIDtoString := 'DENSO WAVE INCORPORATED';

	16#0000078B:
		F_EtherCAT_VendorIDtoString := 'EuroSoft S.r.l.';

	16#0000078C:
		F_EtherCAT_VendorIDtoString := 'University of British Columbia, Faculty of Applied Science, Department of Mechanical Engineering';

	16#0000078D:
		F_EtherCAT_VendorIDtoString := 'REnergy Electric Tianjin Ltd.';

	16#0000078E:
		F_EtherCAT_VendorIDtoString := 'NewYoungSystem Co., Ltd.';

	16#0000078F:
		F_EtherCAT_VendorIDtoString := 'ESA S.p.A.';

	16#00000790:
		F_EtherCAT_VendorIDtoString := 'University of Reading, School of Systems Engineering';

	16#00000791:
		F_EtherCAT_VendorIDtoString := 'KOGANEI CORPORATION';

	16#00000792:
		F_EtherCAT_VendorIDtoString := 'MAZeT GmbH';

	16#00000793:
		F_EtherCAT_VendorIDtoString := 'The University of Nottingham, Faculty of Engineering, Electrical Systems and Optics Research Division';

	16#00000794:
		F_EtherCAT_VendorIDtoString := 'Quanta Storage Inc.';

	16#00000795:
		F_EtherCAT_VendorIDtoString := 'Azbil Taishin Co., Ltd.';

	16#00000796:
		F_EtherCAT_VendorIDtoString := 'Relitech B.V.';

	16#00000797:
		F_EtherCAT_VendorIDtoString := 'DHPC Technologies, Inc.';

	16#00000798:
		F_EtherCAT_VendorIDtoString := 'Jordan Valley Semiconductors Ltd.';

	16#00000799:
		F_EtherCAT_VendorIDtoString := 'MicroCreate System Co., Ltd.';

	16#0000079A:
		F_EtherCAT_VendorIDtoString := 'AB&T S.r.l.';

	16#0000079B:
		F_EtherCAT_VendorIDtoString := 'Medic LLC';

	16#0000079C:
		F_EtherCAT_VendorIDtoString := 'T3LAB - Technology Transfer Team';

	16#0000079D:
		F_EtherCAT_VendorIDtoString := 'Coptonix GmbH';

	16#0000079E:
		F_EtherCAT_VendorIDtoString := 'KARL MAYER STOLL Textilmaschinenfabrik GmbH';

	16#0000079F:
		F_EtherCAT_VendorIDtoString := 'inoson GmbH';

	16#000007A0:
		F_EtherCAT_VendorIDtoString := 'GE Power & Water Distributed Power';

	16#000007A1:
		F_EtherCAT_VendorIDtoString := 'Shanghai Yuanzhi Robot Co., Ltd.';

	16#000007A2:
		F_EtherCAT_VendorIDtoString := 'OYO ELECTRIC CO., LTD.';

	16#000007A3:
		F_EtherCAT_VendorIDtoString := 'Solwit SA';

	16#000007A4:
		F_EtherCAT_VendorIDtoString := 'Jabil Inc.';

	16#000007A5:
		F_EtherCAT_VendorIDtoString := 'Renesas Semiconductor Package & Test Solutions Co., Ltd.';

	16#000007A6:
		F_EtherCAT_VendorIDtoString := 'Technische Universitat Berlin, Fakultat Verkehrs- und Maschinensysteme';

	16#000007A7:
		F_EtherCAT_VendorIDtoString := 'Mettler-Toledo (Changzhou) Precision Instrument Ltd.';

	16#000007A8:
		F_EtherCAT_VendorIDtoString := 'Sentronic International Corp.';

	16#000007A9:
		F_EtherCAT_VendorIDtoString := 'LEAS (Laboratoire delectronique Angelidis et Sarrault)';

	16#000007AA:
		F_EtherCAT_VendorIDtoString := 'MAPNA Electric & Control, Engineering & Manufacturing Co.';

	16#000007AB:
		F_EtherCAT_VendorIDtoString := 'NetTechnix E&P GmbH';

	16#000007AC:
		F_EtherCAT_VendorIDtoString := 'Excelpoint Systems (H.K.) Limited';

	16#000007AD:
		F_EtherCAT_VendorIDtoString := 'Integrated Dynamics Engineering GmbH';

	16#000007AE:
		F_EtherCAT_VendorIDtoString := 'Toho Technology Corporation';

	16#000007AF:
		F_EtherCAT_VendorIDtoString := 'Salvagnini Italia S.p.A.';

	16#000007B0:
		F_EtherCAT_VendorIDtoString := 'Shanghai Triowin Automation Machinery Co., Ltd.';

	16#000007B1:
		F_EtherCAT_VendorIDtoString := 'Hytec Electronics Ltd.';

	16#000007B2:
		F_EtherCAT_VendorIDtoString := 'Xi’an Xiangxun Technology Co., Ltd.';

	16#000007B3:
		F_EtherCAT_VendorIDtoString := 'Schmidiger GmbH';

	16#000007B4:
		F_EtherCAT_VendorIDtoString := 'MASTER LTD.';

	16#000007B5:
		F_EtherCAT_VendorIDtoString := 'Korea University, College of Engineering';

	16#000007B6:
		F_EtherCAT_VendorIDtoString := 'H. Kufferath GmbH Pruf- und Vorrichtungstechnik';

	16#000007B7:
		F_EtherCAT_VendorIDtoString := 'EFTEC Engineering GmbH';

	16#000007B8:
		F_EtherCAT_VendorIDtoString := 'EN2CORE Technology Inc.';

	16#000007B9:
		F_EtherCAT_VendorIDtoString := 'DFC Design, s.r.o.';

	16#000007BA:
		F_EtherCAT_VendorIDtoString := 'FUKUDA CO., LTD.';

	16#000007BB:
		F_EtherCAT_VendorIDtoString := 'Fachhochschule Flensburg';

	16#000007BC:
		F_EtherCAT_VendorIDtoString := 'Karlsruher Institut fur Technologie, IAR, H2T';

	16#000007BD:
		F_EtherCAT_VendorIDtoString := 'Burnon International Ltd.';

	16#000007BE:
		F_EtherCAT_VendorIDtoString := 'Nuova Fima S.P.A.';

	16#000007BF:
		F_EtherCAT_VendorIDtoString := 'Yuban & Co.';

	16#000007C2:
		F_EtherCAT_VendorIDtoString := 'Ricoh Industry Co., Ltd.';

	16#000007C3:
		F_EtherCAT_VendorIDtoString := 'RDC Semiconductor Co., Ltd.';

	16#000007C4:
		F_EtherCAT_VendorIDtoString := 'SETEX Schermuly textile computer GmbH';

	16#000007C5:
		F_EtherCAT_VendorIDtoString := 'elowerk GmbH & Co. KG';

	16#000007C6:
		F_EtherCAT_VendorIDtoString := 'iThemba Laboratory for Accelerator Based Sciences (iThemba LABS)';

	16#000007C7:
		F_EtherCAT_VendorIDtoString := 'Simco (Nederland) B.V.';

	16#000007C8:
		F_EtherCAT_VendorIDtoString := 'CNCSAZAN';

	16#000007C9:
		F_EtherCAT_VendorIDtoString := 'ShiningView Electronic Technology (Shanghai) Co., Ltd.';

	16#000007CA:
		F_EtherCAT_VendorIDtoString := 'Mikysek Engineering';

	16#000007CB:
		F_EtherCAT_VendorIDtoString := 'VICTRON TECHNOLOGY CO., LTD.';

	16#000007CC:
		F_EtherCAT_VendorIDtoString := 'Focke & Co. (GmbH & Co. KG)';

	16#000007CD:
		F_EtherCAT_VendorIDtoString := 'Michigan Scientific Corporation';

	16#000007CE:
		F_EtherCAT_VendorIDtoString := 'ADFweb.com s.r.l.';

	16#000007CF:
		F_EtherCAT_VendorIDtoString := 'Nortion Servo Technology (Beijing) Co., Ltd.';

	16#000007D0:
		F_EtherCAT_VendorIDtoString := 'Akkodis Germany Solutions GmbH';

	16#000007D1:
		F_EtherCAT_VendorIDtoString := 'Zhejiang Synmot Electrical Technology Co., Ltd.';

	16#000007D2:
		F_EtherCAT_VendorIDtoString := 'HK-MnS Co., Ltd.';

	16#000007D3:
		F_EtherCAT_VendorIDtoString := 'Tattile S.r.l.';

	16#000007D4:
		F_EtherCAT_VendorIDtoString := 'ELFIN Pracownia Elektroniki';

	16#000007D5:
		F_EtherCAT_VendorIDtoString := 'Bimba Manufacturing Company';

	16#000007D6:
		F_EtherCAT_VendorIDtoString := 'Winsonic Electronics Co., Ltd.';

	16#000007D7:
		F_EtherCAT_VendorIDtoString := 'DIMETIX AG';

	16#000007D8:
		F_EtherCAT_VendorIDtoString := 'GENETEC CORPORATION';

	16#000007D9:
		F_EtherCAT_VendorIDtoString := 'Tianjin Hengxin Chuangyuan Science & Technology Co., Ltd.';

	16#000007DA:
		F_EtherCAT_VendorIDtoString := 'SFA Engineering Corp.';

	16#000007DB:
		F_EtherCAT_VendorIDtoString := 'Opticon Inc.';

	16#000007DC:
		F_EtherCAT_VendorIDtoString := 'NPN Co., Ltd.';

	16#000007DD:
		F_EtherCAT_VendorIDtoString := 'Wuhan Maxsine Electric Co., Ltd.';

	16#000007DF:
		F_EtherCAT_VendorIDtoString := 'Concept Overdrive Inc.';

	16#000007E0:
		F_EtherCAT_VendorIDtoString := 'HETRONIK GmbH';

	16#000007E2:
		F_EtherCAT_VendorIDtoString := 'JBT Corporation';

	16#000007E3:
		F_EtherCAT_VendorIDtoString := 'Technische Universitat Dresden, Fakultat Elektrotechnik und Informationstechnik';

	16#000007E4:
		F_EtherCAT_VendorIDtoString := 'DAJO Solutions Ltd.';

	16#000007E5:
		F_EtherCAT_VendorIDtoString := 'Criterion NDT, Inc.';

	16#000007E6:
		F_EtherCAT_VendorIDtoString := 'Quanzhou Sangchuan Electric Equipment Co., Ltd.';

	16#000007E7:
		F_EtherCAT_VendorIDtoString := 'DATA TECNO Co. Ltd.';

	16#000007E8:
		F_EtherCAT_VendorIDtoString := 'Rainbow Springs Pvt Ltd.';

	16#000007E9:
		F_EtherCAT_VendorIDtoString := 'Renu Electronics Pvt. Ltd.';

	16#000007EA:
		F_EtherCAT_VendorIDtoString := 'Max-Planck-Institut fur biologische Kybernetik, Abteilung Wahrnehmung, Kognition und Handlung';

	16#000007EB:
		F_EtherCAT_VendorIDtoString := 'Intelligent Automation Equipment (Zhuhai) Co., Ltd.';

	16#000007EC:
		F_EtherCAT_VendorIDtoString := 'SCREEN Holdings Co., Ltd.';

	16#000007ED:
		F_EtherCAT_VendorIDtoString := 'Sysmex Corporation';

	16#000007EE:
		F_EtherCAT_VendorIDtoString := 'ASM Japan K.K.';

	16#000007EF:
		F_EtherCAT_VendorIDtoString := 'IMAGO Technologies GmbH';

	16#000007F0:
		F_EtherCAT_VendorIDtoString := 'Happiest Minds Technologies Private Limited';

	16#000007F1:
		F_EtherCAT_VendorIDtoString := 'Open Control System Technology Co. Ltd.';

	16#000007F2:
		F_EtherCAT_VendorIDtoString := 'University of Seoul, College of Engineering';

	16#000007F3:
		F_EtherCAT_VendorIDtoString := 'ULVAC, Inc.';

	16#000007F4:
		F_EtherCAT_VendorIDtoString := 'Meliora Scientific Inc.';

	16#000007F5:
		F_EtherCAT_VendorIDtoString := 'Toshiba Corporation';

	16#000007F6:
		F_EtherCAT_VendorIDtoString := 'Schnell Spa';

	16#000007F7:
		F_EtherCAT_VendorIDtoString := 'Industrial Technology Research Institute (ITRI)';

	16#000007F8:
		F_EtherCAT_VendorIDtoString := '4PICO BV';

	16#000007F9:
		F_EtherCAT_VendorIDtoString := 'AVL SET GmbH';

	16#000007FA:
		F_EtherCAT_VendorIDtoString := 'CHANGNAM I.N.T. LTD.';

	16#000007FB:
		F_EtherCAT_VendorIDtoString := 'Shanghai Ruking Technology Co., Ltd.';

	16#000007FC:
		F_EtherCAT_VendorIDtoString := 'META Srl';

	16#000007FD:
		F_EtherCAT_VendorIDtoString := 'GHM Messtechnik GmbH';

	16#000007FF:
		F_EtherCAT_VendorIDtoString := 'Xihua University';

	16#00000800:
		F_EtherCAT_VendorIDtoString := 'Stratus Automation Sdn. Bhd.';

	16#00000801:
		F_EtherCAT_VendorIDtoString := 'OTSL Inc.';

	16#00000802:
		F_EtherCAT_VendorIDtoString := 'Aromasoft Corp.';

	16#00000803:
		F_EtherCAT_VendorIDtoString := 'Bobst Mex SA';

	16#00000804:
		F_EtherCAT_VendorIDtoString := 'Beijing Powerbeck Automation Technology CO., LTD.';

	16#00000805:
		F_EtherCAT_VendorIDtoString := 'TESSERA TECHNOLOGY INC.';

	16#00000806:
		F_EtherCAT_VendorIDtoString := 'JWiesemann.com - Dr. Joachim Wiesemann';

	16#00000807:
		F_EtherCAT_VendorIDtoString := 'Istanbul Ulasim San Tic. A.S.';

	16#00000808:
		F_EtherCAT_VendorIDtoString := 'ProPhotonix (Irl) Ltd.';

	16#00000809:
		F_EtherCAT_VendorIDtoString := 'B.I.N.S.S Datennetze und Gefahrenmeldesysteme GmbH';

	16#0000080A:
		F_EtherCAT_VendorIDtoString := 'University "Stefan cel Mare" Suceava, Electrical Engineering and Computer Science';

	16#0000080B:
		F_EtherCAT_VendorIDtoString := 'Modrol Electric CO., Ltd.';

	16#0000080C:
		F_EtherCAT_VendorIDtoString := 'OBS Korea Co.,Ltd';

	16#0000080D:
		F_EtherCAT_VendorIDtoString := 'Shanghai Jiao Tong University, School of Mechanical Engineering';

	16#0000080E:
		F_EtherCAT_VendorIDtoString := 'TEAM ELECTRONICS GmbH';

	16#0000080F:
		F_EtherCAT_VendorIDtoString := 'Southwest University of Science and Technology (SWUST) National University Science Park';

	16#00000810:
		F_EtherCAT_VendorIDtoString := 'TDK-Lambda Americas Inc.';

	16#00000811:
		F_EtherCAT_VendorIDtoString := 'Ta Liang Technology Co. Ltd.';

	16#00000812:
		F_EtherCAT_VendorIDtoString := 'CCS Inc.';

	16#00000813:
		F_EtherCAT_VendorIDtoString := 'adaptronic Pruftechnik GmbH';

	16#00000814:
		F_EtherCAT_VendorIDtoString := 'TOHO Electronics Inc.';

	16#00000815:
		F_EtherCAT_VendorIDtoString := 'VMek Group LLC (dba VMek Sorting Technology)';

	16#00000816:
		F_EtherCAT_VendorIDtoString := 'CKD Nikki Denso Co., Ltd.';

	16#00000817:
		F_EtherCAT_VendorIDtoString := 'Systematic Consulting Group, Inc.';

	16#00000818:
		F_EtherCAT_VendorIDtoString := 'PERITEC Corporation';

	16#00000819:
		F_EtherCAT_VendorIDtoString := 'Bachmann Technology GmbH & Co. KG';

	16#0000081A:
		F_EtherCAT_VendorIDtoString := 'BMK electronic solutions GmbH & Co. KG';

	16#0000081B:
		F_EtherCAT_VendorIDtoString := 'TECO Electric & Machinery Co., Ltd.';

	16#0000081C:
		F_EtherCAT_VendorIDtoString := 'Mechtronic Industries Ltd.';

	16#0000081D:
		F_EtherCAT_VendorIDtoString := 'Mernok Elektronik (Pty) Ltd.';

	16#0000081E:
		F_EtherCAT_VendorIDtoString := 'Universitat Bremen, Institut fur elektrische Antriebe, Leistungselektronik und Bauelemente';

	16#0000081F:
		F_EtherCAT_VendorIDtoString := 'Hydro-Quebec Research Institute';

	16#00000820:
		F_EtherCAT_VendorIDtoString := 'GEMTEC Laseroptische Systeme GmbH';

	16#00000821:
		F_EtherCAT_VendorIDtoString := 'SINTEF Raufoss Manufacturing AS';

	16#00000822:
		F_EtherCAT_VendorIDtoString := 'Advanced Manufacturing Engineering Technologies Inc.';

	16#00000823:
		F_EtherCAT_VendorIDtoString := 'Levitronix GmbH';

	16#00000825:
		F_EtherCAT_VendorIDtoString := 'Dipl.-Ing. Carsten Spie Softwareentwicklung';

	16#00000826:
		F_EtherCAT_VendorIDtoString := 'Reivax S/A Automacao e Controle';

	16#00000827:
		F_EtherCAT_VendorIDtoString := 'Lappeenranta University of Technology (LUT), School of Energy Systems, Electrical Engineering';

	16#00000828:
		F_EtherCAT_VendorIDtoString := 'TOTANI CORPORATION';

	16#00000829:
		F_EtherCAT_VendorIDtoString := 'SERAD S.A.S.';

	16#0000082A:
		F_EtherCAT_VendorIDtoString := 'ITW Dynatec GmbH';

	16#0000082B:
		F_EtherCAT_VendorIDtoString := 'Hochschule Emden/Leer, Fachbereich Technik';

	16#0000082C:
		F_EtherCAT_VendorIDtoString := 'JFControl Co., Ltd.';

	16#0000082D:
		F_EtherCAT_VendorIDtoString := 'SAEL srl';

	16#0000082E:
		F_EtherCAT_VendorIDtoString := 'Beckman Coulter Biomedical GmbH';

	16#0000082F:
		F_EtherCAT_VendorIDtoString := 'Walter Maschinenbau GmbH';

	16#00000830:
		F_EtherCAT_VendorIDtoString := 'Alterface s.a.';

	16#00000831:
		F_EtherCAT_VendorIDtoString := 'Lectronix, Inc.';

	16#00000832:
		F_EtherCAT_VendorIDtoString := 'HOKUYO AUTOMATIC CO., LTD.';

	16#00000833:
		F_EtherCAT_VendorIDtoString := 'Shanghai Empower Technologies Co., Ltd.';

	16#00000834:
		F_EtherCAT_VendorIDtoString := 'Thyracont Vacuum Instruments GmbH';

	16#00000835:
		F_EtherCAT_VendorIDtoString := 'OMAX Corporation';

	16#00000836:
		F_EtherCAT_VendorIDtoString := 'TOX PRESSOTECHNIK SE & Co. KG';

	16#00000837:
		F_EtherCAT_VendorIDtoString := 'National Chiao Tung University, College of Electrical and Computer Engineering, Department of Electrical Engineering';

	16#00000838:
		F_EtherCAT_VendorIDtoString := 'Inspiro BV';

	16#00000839:
		F_EtherCAT_VendorIDtoString := 'Maxcess International';

	16#0000083A:
		F_EtherCAT_VendorIDtoString := 'Chell Instruments Ltd.';

	16#0000083B:
		F_EtherCAT_VendorIDtoString := 'FUJI CORPORATION';

	16#0000083C:
		F_EtherCAT_VendorIDtoString := 'NIDEC INSTRUMENTS CORPORATION';

	16#0000083D:
		F_EtherCAT_VendorIDtoString := 'Shizuoka Oki Electric Co., Ltd.';

	16#0000083E:
		F_EtherCAT_VendorIDtoString := 'Frencken America Inc.';

	16#0000083F:
		F_EtherCAT_VendorIDtoString := 'Granite Devices Oy';

	16#00000840:
		F_EtherCAT_VendorIDtoString := 'SANEZOO EUROPE s.r.o.';

	16#00000842:
		F_EtherCAT_VendorIDtoString := 'AGILiCOM SARL';

	16#00000843:
		F_EtherCAT_VendorIDtoString := 'TRUMPF Photonic Components GmbH';

	16#00000844:
		F_EtherCAT_VendorIDtoString := 'KLA Corporation';

	16#00000845:
		F_EtherCAT_VendorIDtoString := 'Meidensha Corporation';

	16#00000849:
		F_EtherCAT_VendorIDtoString := 'Rolls-Royce Nuclear Services';

	16#0000084A:
		F_EtherCAT_VendorIDtoString := 'University of West Bohemia, Faculty of Applied Sciences';

	16#0000084B:
		F_EtherCAT_VendorIDtoString := 'Korea Electrotechnology Research Institute (KERI)';

	16#0000084C:
		F_EtherCAT_VendorIDtoString := 'MPI Corporation';

	16#0000084D:
		F_EtherCAT_VendorIDtoString := 'Roders GmbH';

	16#0000084E:
		F_EtherCAT_VendorIDtoString := 'Melec Inc.';

	16#0000084F:
		F_EtherCAT_VendorIDtoString := 'Mianyang Weibo Electronic Co., Ltd.';

	16#00000851:
		F_EtherCAT_VendorIDtoString := 'Wuhan Huazhong Numerical Control Co., Ltd.';

	16#00000852:
		F_EtherCAT_VendorIDtoString := 'Datalogic S.r.l.';

	16#00000853:
		F_EtherCAT_VendorIDtoString := 'Tri-Tek Corp.';

	16#00000855:
		F_EtherCAT_VendorIDtoString := 'YUHENG OPTICS CO.,LTD (Changchun)';

	16#00000856:
		F_EtherCAT_VendorIDtoString := 'ETH-messtechnik gmbh';

	16#00000857:
		F_EtherCAT_VendorIDtoString := 'JTEKT CORPORATION';

	16#00000858:
		F_EtherCAT_VendorIDtoString := 'ergo: elektronik GmbH';

	16#00000859:
		F_EtherCAT_VendorIDtoString := 'Engineerdream Co., Ltd.';

	16#0000085A:
		F_EtherCAT_VendorIDtoString := 'Samsung Electronics Co. Ltd.';

	16#0000085B:
		F_EtherCAT_VendorIDtoString := 'KSJ Co. Ltd.';

	16#0000085C:
		F_EtherCAT_VendorIDtoString := 'Messer Cutting Systems GmbH';

	16#0000085D:
		F_EtherCAT_VendorIDtoString := 'Krones AG';

	16#0000085F:
		F_EtherCAT_VendorIDtoString := 'Northwestern Polytechnical University, School of Power&Energy, Department of Power Control and Test';

	16#00000860:
		F_EtherCAT_VendorIDtoString := 'Blackbird Robotersysteme GmbH';

	16#00000861:
		F_EtherCAT_VendorIDtoString := 'Mitsuba Corporation';

	16#00000863:
		F_EtherCAT_VendorIDtoString := 'Foshan Shunde Gatherwin Information Technology Co., Ltd.';

	16#00000864:
		F_EtherCAT_VendorIDtoString := 'duagon Germany GmbH';

	16#00000865:
		F_EtherCAT_VendorIDtoString := 'Thermo Fisher Scientific Oy';

	16#00000866:
		F_EtherCAT_VendorIDtoString := 'Pyramid Technical Consultants';

	16#00000867:
		F_EtherCAT_VendorIDtoString := 'Verity Instruments, Inc.';

	16#00000868:
		F_EtherCAT_VendorIDtoString := 'KAI PLUS TECHNOLOGY CO., LTD.';

	16#00000869:
		F_EtherCAT_VendorIDtoString := 'Texas A&M University at Qatar, Electrical & Computer Engineering';

	16#0000086A:
		F_EtherCAT_VendorIDtoString := 'FPT Motorenforschung AG';

	16#0000086B:
		F_EtherCAT_VendorIDtoString := 'Industries Machinex Inc.';

	16#0000086C:
		F_EtherCAT_VendorIDtoString := 'Shanghai Rising Digital Co.,Ltd.';

	16#0000086D:
		F_EtherCAT_VendorIDtoString := 'SICK OPTEX CO., LTD.';

	16#0000086E:
		F_EtherCAT_VendorIDtoString := 'Laserline GmbH';

	16#0000086F:
		F_EtherCAT_VendorIDtoString := 'Xpress Precision Engineering B.V.';

	16#00000870:
		F_EtherCAT_VendorIDtoString := 'ELECTRA S.p.A.';

	16#00000871:
		F_EtherCAT_VendorIDtoString := 'Magnescale Co., Ltd.';

	16#00000872:
		F_EtherCAT_VendorIDtoString := 'Hitachi Kokusai Electric Inc.';

	16#00000873:
		F_EtherCAT_VendorIDtoString := 'Hangzhou Jingwei Automation Co., Ltd.';

	16#00000874:
		F_EtherCAT_VendorIDtoString := 'Shanghai LYNUC CNC Technology Co., Ltd.';

	16#00000875:
		F_EtherCAT_VendorIDtoString := 'ATLAS ELEKTRONIK GmbH';

	16#00000876:
		F_EtherCAT_VendorIDtoString := 'EDAC Electronics Technology (Hangzhou) Co., Ltd.';

	16#00000877:
		F_EtherCAT_VendorIDtoString := 'MYCOM, INC.';

	16#00000878:
		F_EtherCAT_VendorIDtoString := 'ElectroCraft, Inc.';

	16#00000879:
		F_EtherCAT_VendorIDtoString := 'Foxconn Technology Group';

	16#0000087A:
		F_EtherCAT_VendorIDtoString := 'Qinhuangdao Boostsolar Photovoltatic Equipment Co.,Ltd.';

	16#0000087B:
		F_EtherCAT_VendorIDtoString := 'Chinese Academy of Sciences, Shenyang Institute of Automation (SIA)';

	16#0000087C:
		F_EtherCAT_VendorIDtoString := 'Deere & Company';

	16#0000087D:
		F_EtherCAT_VendorIDtoString := 'Leibniz Universitat Hannover, Institut fur Mechatronische Systeme (IMES)';

	16#0000087F:
		F_EtherCAT_VendorIDtoString := 'ELTRO Gesellschaft fur Elektrotechnik mbH';

	16#00000880:
		F_EtherCAT_VendorIDtoString := 'UK Grid Solutions Limited';

	16#00000881:
		F_EtherCAT_VendorIDtoString := 'Control Gaging, Inc.';

	16#00000882:
		F_EtherCAT_VendorIDtoString := 'Trilix Engineering AG';

	16#00000883:
		F_EtherCAT_VendorIDtoString := 'HFE professionelle Studiotechnik GmbH';

	16#00000884:
		F_EtherCAT_VendorIDtoString := 'HMT Co., Ltd.';

	16#00000885:
		F_EtherCAT_VendorIDtoString := 'SCHNIER Elektrostatik GmbH';

	16#00000886:
		F_EtherCAT_VendorIDtoString := 'Wuhan HuaGong Laser Engineering Co.,Ltd.';

	16#00000888:
		F_EtherCAT_VendorIDtoString := 'Zhejiang Keqiang Intelligent Control System Co., Ltd.';

	16#00000889:
		F_EtherCAT_VendorIDtoString := 'Impedans Ltd.';

	16#0000088A:
		F_EtherCAT_VendorIDtoString := 'Chinese Academy of Sciences, Institute of Automation';

	16#0000088B:
		F_EtherCAT_VendorIDtoString := 'GCCAlliance Inc.';

	16#0000088C:
		F_EtherCAT_VendorIDtoString := 'Interface Corporation';

	16#0000088D:
		F_EtherCAT_VendorIDtoString := 'NEC Platforms, Ltd.';

	16#0000088E:
		F_EtherCAT_VendorIDtoString := 'Shenyang Piotech Co., Ltd.';

	16#0000088F:
		F_EtherCAT_VendorIDtoString := 'TQ-Systems GmbH';

	16#00000890:
		F_EtherCAT_VendorIDtoString := 'Shanghai Panelmate Electronics Co., Ltd.';

	16#00000891:
		F_EtherCAT_VendorIDtoString := 'Haute Ecole Arc Ingenierie';

	16#00000892:
		F_EtherCAT_VendorIDtoString := 'Korea Institute of Industrial Technology - KITECH';

	16#00000893:
		F_EtherCAT_VendorIDtoString := 'CETA Testsysteme GmbH';

	16#00000895:
		F_EtherCAT_VendorIDtoString := 'STEP Corporation';

	16#00000896:
		F_EtherCAT_VendorIDtoString := 'Dalian Guangyang Science & Technology Group Co., Ltd.';

	16#00000897:
		F_EtherCAT_VendorIDtoString := 'Hermes Microvision, Inc.';

	16#00000898:
		F_EtherCAT_VendorIDtoString := 'Kawasaki Heavy Industries, Ltd., Robot Division';

	16#00000899:
		F_EtherCAT_VendorIDtoString := 'ELCO Industry Automation AG';

	16#0000089A:
		F_EtherCAT_VendorIDtoString := 'Neuromeka';

	16#0000089D:
		F_EtherCAT_VendorIDtoString := 'SEMES Co., Ltd.';

	16#0000089E:
		F_EtherCAT_VendorIDtoString := 'FEV SA';

	16#0000089F:
		F_EtherCAT_VendorIDtoString := 'Plasmart Inc.';

	16#000008A0:
		F_EtherCAT_VendorIDtoString := 'DRESCHER Industrieelektronik GmbH';

	16#000008A1:
		F_EtherCAT_VendorIDtoString := 'MK  SYSTEM CO.,LTD';

	16#000008A2:
		F_EtherCAT_VendorIDtoString := 'bebro electronic GmbH';

	16#000008A3:
		F_EtherCAT_VendorIDtoString := 'MC-monitoring SA';

	16#000008A4:
		F_EtherCAT_VendorIDtoString := 'Variable Message Signs (a trading division of Hill & Smith Ltd)';

	16#000008A5:
		F_EtherCAT_VendorIDtoString := 'Dukane Corporation - Intelligent Assembly Solutions';

	16#000008A6:
		F_EtherCAT_VendorIDtoString := 'Mecatronix GmbH';

	16#000008A7:
		F_EtherCAT_VendorIDtoString := 'Prima Power Laserdyne LLC';

	16#000008A8:
		F_EtherCAT_VendorIDtoString := 'ISOCOMP srl';

	16#000008A9:
		F_EtherCAT_VendorIDtoString := 'Shinko Shoji Co.,Ltd.';

	16#000008AA:
		F_EtherCAT_VendorIDtoString := 'ASEC International Corporation';

	16#000008AB:
		F_EtherCAT_VendorIDtoString := 'RTC Electronics Ltd.';

	16#000008AC:
		F_EtherCAT_VendorIDtoString := 'Entegris, Inc.';

	16#000008AD:
		F_EtherCAT_VendorIDtoString := 'ASEM S.r.l.';

	16#000008AE:
		F_EtherCAT_VendorIDtoString := 'Beijing Agie Charmilles Industrial Electronics Co., Ltd.';

	16#000008AF:
		F_EtherCAT_VendorIDtoString := 'Zhengzhou Changhe Electronic Engineering Co., Ltd.';

	16#000008B0:
		F_EtherCAT_VendorIDtoString := 'Leister Technologies AG';

	16#000008B2:
		F_EtherCAT_VendorIDtoString := 'SAGINOMIYA SEISAKUSHO, INC.';

	16#000008B3:
		F_EtherCAT_VendorIDtoString := 'LNC Technology Co., Ltd.';

	16#000008B4:
		F_EtherCAT_VendorIDtoString := 'Guangdong ELESY Electric CO., LTD.';

	16#000008B5:
		F_EtherCAT_VendorIDtoString := 'Newtouch Electronics (Shanghai) Co.,Ltd.';

	16#000008B6:
		F_EtherCAT_VendorIDtoString := 'TOYO AUTOMATION CO., LTD.';

	16#000008B7:
		F_EtherCAT_VendorIDtoString := 'Universite de Bretagne-Sud';

	16#000008B8:
		F_EtherCAT_VendorIDtoString := 'Shenzhen Zhiyou Battery Integration Technology Co., Ltd.';

	16#000008B9:
		F_EtherCAT_VendorIDtoString := 'Malema Engineering Corporation';

	16#000008BB:
		F_EtherCAT_VendorIDtoString := 'Ricoh Industrial Solutions Inc.';

	16#000008BC:
		F_EtherCAT_VendorIDtoString := 'Tri-City X-ray, LLC';

	16#000008BD:
		F_EtherCAT_VendorIDtoString := 'Rutronik Elektronische Bauelemente GmbH';

	16#000008BE:
		F_EtherCAT_VendorIDtoString := 'SANEI HYTECHS VIETNAM Co.,Ltd.';

	16#000008BF:
		F_EtherCAT_VendorIDtoString := 'Delixi (Hangzhou) Inverter Co.,LTD.';

	16#000008C0:
		F_EtherCAT_VendorIDtoString := 'RITZ Co., Ltd.';

	16#000008C1:
		F_EtherCAT_VendorIDtoString := 'Ricoh Company, Ltd.';

	16#000008C2:
		F_EtherCAT_VendorIDtoString := 'TAE Antriebstechnik GmbH';

	16#000008C3:
		F_EtherCAT_VendorIDtoString := 'Fontys University of Applied Sciences';

	16#000008C4:
		F_EtherCAT_VendorIDtoString := 'Hangzhou Riding Control Technology Co., Ltd.';

	16#000008C5:
		F_EtherCAT_VendorIDtoString := 'Atlas Copco Industrial Technique AB';

	16#000008C6:
		F_EtherCAT_VendorIDtoString := 'Mindtribe Product Engineering, Inc.';

	16#000008C7:
		F_EtherCAT_VendorIDtoString := 'Centre de recherche industrielle du Quebec (CRIQ)';

	16#000008C8:
		F_EtherCAT_VendorIDtoString := 'Elster GmbH';

	16#000008C9:
		F_EtherCAT_VendorIDtoString := 'Panasonic Industrial Devices Systems and Technology Co., Ltd.';

	16#000008CA:
		F_EtherCAT_VendorIDtoString := 'STV Electronic GmbH & Co. KG';

	16#000008CB:
		F_EtherCAT_VendorIDtoString := 'Hentschel System GmbH';

	16#000008CC:
		F_EtherCAT_VendorIDtoString := 'Gree Electric Appliances, Inc. of Zhuhai';

	16#000008CD:
		F_EtherCAT_VendorIDtoString := 'Futurestar Corp.';

	16#000008CE:
		F_EtherCAT_VendorIDtoString := 'PARA-ENT CO.,LTD.';

	16#000008CF:
		F_EtherCAT_VendorIDtoString := 'SIASUN CO., LTD.';

	16#000008D0:
		F_EtherCAT_VendorIDtoString := 'WFE Technology Corporation';

	16#000008D1:
		F_EtherCAT_VendorIDtoString := 'driveXpert GmbH';

	16#000008D2:
		F_EtherCAT_VendorIDtoString := 'Universitat zu Lubeck, Institut fur Medizinische Elektrotechnik';

	16#000008D3:
		F_EtherCAT_VendorIDtoString := 'SCE s.r.l. Elettronica per Automazioni';

	16#000008D4:
		F_EtherCAT_VendorIDtoString := 'Branson Ultrasonics Corporation';

	16#000008D5:
		F_EtherCAT_VendorIDtoString := 'Rolls-Royce@NTU Corporate Lab';

	16#000008D6:
		F_EtherCAT_VendorIDtoString := 'Guilin Stars Science and Technology CO., LTD.';

	16#000008D7:
		F_EtherCAT_VendorIDtoString := 'Ace Designers Limited';

	16#000008D8:
		F_EtherCAT_VendorIDtoString := 'Biochar Now LLC';

	16#000008D9:
		F_EtherCAT_VendorIDtoString := 'Varian Medical Systems Inc.';

	16#000008DA:
		F_EtherCAT_VendorIDtoString := 'DAMEDICS GmbH';

	16#000008DB:
		F_EtherCAT_VendorIDtoString := 'EnergopromAvtomatizaciya LLC';

	16#000008DC:
		F_EtherCAT_VendorIDtoString := 'MicroSure B.V.';

	16#000008DE:
		F_EtherCAT_VendorIDtoString := 'Finisar SHG Inc.';

	16#000008DF:
		F_EtherCAT_VendorIDtoString := 'PLANET Technology Corporation';

	16#000008E0:
		F_EtherCAT_VendorIDtoString := 'PEES Components GmbH';

	16#000008E1:
		F_EtherCAT_VendorIDtoString := 'Belden Deutschland GmbH';

	16#000008E2:
		F_EtherCAT_VendorIDtoString := 'NACHI-FUJIKOSHI CORP.';

	16#000008E3:
		F_EtherCAT_VendorIDtoString := 'K. A. Schmersal GmbH & Co. KG';

	16#000008E4:
		F_EtherCAT_VendorIDtoString := 'Radic Technologies, Inc.';

	16#000008E5:
		F_EtherCAT_VendorIDtoString := 'Weightpack S.r.l.';

	16#000008E6:
		F_EtherCAT_VendorIDtoString := 'BS2 MULTIDATA GmbH';

	16#000008E7:
		F_EtherCAT_VendorIDtoString := 'Sumitomo Heavy Industries, Ltd.';

	16#000008E8:
		F_EtherCAT_VendorIDtoString := 'Micro-Controle Spectra-Physics S.A.';

	16#000008E9:
		F_EtherCAT_VendorIDtoString := 'Apptronik Inc.';

	16#000008EA:
		F_EtherCAT_VendorIDtoString := 'Dr.-Ing. S. Haumann Industrieelektronik';

	16#000008EB:
		F_EtherCAT_VendorIDtoString := 'Great River Electronics, Inc.';

	16#000008EC:
		F_EtherCAT_VendorIDtoString := 'Eltra S.p.a. Unipersonale';

	16#000008ED:
		F_EtherCAT_VendorIDtoString := 'SINOBONDER Co., Ltd.';

	16#000008EE:
		F_EtherCAT_VendorIDtoString := 'ROBOTOUS Co., Ltd.';

	16#000008EF:
		F_EtherCAT_VendorIDtoString := 'Tianjin Sentinel Electronics Co.,Ltd.';

	16#000008F0:
		F_EtherCAT_VendorIDtoString := 'IZOVAC LTD';

	16#000008F1:
		F_EtherCAT_VendorIDtoString := 'Technical University of Kosice, Faculty of Electrical Engineering and Informatics';

	16#000008F2:
		F_EtherCAT_VendorIDtoString := 'SANMEI ELECTRONICS Co., Ltd.';

	16#000008F3:
		F_EtherCAT_VendorIDtoString := 'EA Elektro-Automatik GmbH';

	16#000008F4:
		F_EtherCAT_VendorIDtoString := 'Dynamic Motion Italia S.r.l.';

	16#000008F5:
		F_EtherCAT_VendorIDtoString := 'OOO PKF Ersted';

	16#000008F6:
		F_EtherCAT_VendorIDtoString := 'SHANGHAI MAIHONG ELECTRONIC TECHNOLOGY CO.LTD';

	16#000008F7:
		F_EtherCAT_VendorIDtoString := 'China Electronics Harvest Technology Co.,Ltd.';

	16#000008F8:
		F_EtherCAT_VendorIDtoString := 'Advanced Scientific Technology & Management Research Institute of Kyoto (ASTEM RI)';

	16#000008F9:
		F_EtherCAT_VendorIDtoString := 'Mini Motor srl';

	16#000008FA:
		F_EtherCAT_VendorIDtoString := 'BitifEye Digital Test Solutions GmbH';

	16#000008FB:
		F_EtherCAT_VendorIDtoString := 'IBIS Computer Pty Ltd';

	16#000008FC:
		F_EtherCAT_VendorIDtoString := 'Hanbit Micro Inc.';

	16#000008FD:
		F_EtherCAT_VendorIDtoString := 'TATEYAMA KAGAKU MODULE TECHNOLOGY CO., LTD.';

	16#000008FF:
		F_EtherCAT_VendorIDtoString := 'Aone Co.,Ltd';

	16#00000900:
		F_EtherCAT_VendorIDtoString := 'Shanghai Capital Numerical Control Co., Ltd.';

	16#00000901:
		F_EtherCAT_VendorIDtoString := 'Bose Corporation';

	16#00000902:
		F_EtherCAT_VendorIDtoString := 'Flow Devices and Systems, Inc.';

	16#00000904:
		F_EtherCAT_VendorIDtoString := 'Anritsu Engineering Co., Ltd.';

	16#00000905:
		F_EtherCAT_VendorIDtoString := 'NUTPOR BREADS, UNIPESSOAL LDA.';

	16#00000906:
		F_EtherCAT_VendorIDtoString := 'Emerson SolaHD (a division of Appleton GRP LLC dba Appleton Group)';

	16#00000907:
		F_EtherCAT_VendorIDtoString := 'modusoft GmbH';

	16#00000908:
		F_EtherCAT_VendorIDtoString := 'Sichuan MK Servo Technology';

	16#00000909:
		F_EtherCAT_VendorIDtoString := 'Shanghai Intron Electronics Co.,Ltd.';

	16#0000090A:
		F_EtherCAT_VendorIDtoString := 'Jimei University, College of Information Engineering';

	16#0000090C:
		F_EtherCAT_VendorIDtoString := 'CORE CORPORATION';

	16#0000090D:
		F_EtherCAT_VendorIDtoString := 'H.I.B Systemtechnik GmbH';

	16#0000090E:
		F_EtherCAT_VendorIDtoString := 'Nova Fabrica Ltd.';

	16#0000090F:
		F_EtherCAT_VendorIDtoString := 'ROTA TEKNIK MAKINA SAN. ve TIC. A.S.';

	16#00000910:
		F_EtherCAT_VendorIDtoString := 'Bird Technologies Group, Inc.';

	16#00000911:
		F_EtherCAT_VendorIDtoString := 'SHENZHEN VMMORE CTRL&TECH CO., LTD';

	16#00000912:
		F_EtherCAT_VendorIDtoString := 'Leibniz Universitat Hannover, Fakultat fur Elektrotechnik und Informatik';

	16#00000913:
		F_EtherCAT_VendorIDtoString := 'Motion Control Products Ltd.';

	16#00000914:
		F_EtherCAT_VendorIDtoString := 'Saft S.A.S.';

	16#00000915:
		F_EtherCAT_VendorIDtoString := 'Star Denshi Co.,Ltd.';

	16#00000916:
		F_EtherCAT_VendorIDtoString := 'MARPOSS S.p.A.';

	16#00000917:
		F_EtherCAT_VendorIDtoString := 'China Orient Institute of Noise & Vibration';

	16#00000918:
		F_EtherCAT_VendorIDtoString := 'Cosys Inc.';

	16#00000919:
		F_EtherCAT_VendorIDtoString := 'Shenzhen Vector Automation Technology Co., Lt';

	16#0000091B:
		F_EtherCAT_VendorIDtoString := 'INTRAVIS GmbH';

	16#0000091C:
		F_EtherCAT_VendorIDtoString := 'Drobak Unlimited Co.';

	16#0000091D:
		F_EtherCAT_VendorIDtoString := 'Technische Hochschule Nurnberg Georg Simon Ohm';

	16#0000091E:
		F_EtherCAT_VendorIDtoString := 'Zenitron Corporation';

	16#0000091F:
		F_EtherCAT_VendorIDtoString := 'Wuhan Endeavor Intelligent Machine Co., Ltd.';

	16#00000920:
		F_EtherCAT_VendorIDtoString := 'LEADJECK AUTOMATION CO., LTD.';

	16#00000922:
		F_EtherCAT_VendorIDtoString := 'Fujian Raynen Technology Co., Ltd.';

	16#00000923:
		F_EtherCAT_VendorIDtoString := 'Demcon Advanced Mechatronics B.V.';

	16#00000924:
		F_EtherCAT_VendorIDtoString := 'serva transport systems GmbH';

	16#00000925:
		F_EtherCAT_VendorIDtoString := 'Shenyang Neusoft Medical Systems Co., Ltd.';

	16#00000926:
		F_EtherCAT_VendorIDtoString := 'Ruhr-Universitat Bochum';

	16#00000927:
		F_EtherCAT_VendorIDtoString := 'Banner Engineering Corporation';

	16#00000928:
		F_EtherCAT_VendorIDtoString := 'Ningbo Yunsheng Edrive Technologies Co., Ltd';

	16#00000929:
		F_EtherCAT_VendorIDtoString := 'Guangdong Topstar Technology Co., Ltd.';

	16#0000092A:
		F_EtherCAT_VendorIDtoString := 'Evinsys LLC';

	16#0000092B:
		F_EtherCAT_VendorIDtoString := 'Shenzhen Huacheng Industrial Control Co., Ltd.';

	16#0000092C:
		F_EtherCAT_VendorIDtoString := 'Mondragon Unibertsitatea';

	16#0000092D:
		F_EtherCAT_VendorIDtoString := 'Katholieke Hogeschool Vives (VIVES)';

	16#0000092E:
		F_EtherCAT_VendorIDtoString := 'Ekso Bionics Inc.';

	16#0000092F:
		F_EtherCAT_VendorIDtoString := 'Kaufman & Robinson Inc.';

	16#00000930:
		F_EtherCAT_VendorIDtoString := 'KSM-ELECTRONIC GmbH';

	16#00000931:
		F_EtherCAT_VendorIDtoString := 'Shenzhen Blue Dynamics Precision Co., Ltd.';

	16#00000932:
		F_EtherCAT_VendorIDtoString := 'Technical & Try Co.,Ltd';

	16#00000935:
		F_EtherCAT_VendorIDtoString := 'MAXCOM Co.,Ltd.';

	16#00000936:
		F_EtherCAT_VendorIDtoString := 'National NC System Engineering Research Center';

	16#00000937:
		F_EtherCAT_VendorIDtoString := 'Ryoei Technica Corporation';

	16#00000938:
		F_EtherCAT_VendorIDtoString := 'Schaeffler Technologies AG & Co. KG';

	16#00000939:
		F_EtherCAT_VendorIDtoString := 'NTS-Group';

	16#0000093A:
		F_EtherCAT_VendorIDtoString := 'Alicat Scientific, Inc.';

	16#0000093B:
		F_EtherCAT_VendorIDtoString := 'Tekt Industries Pty. Ltd.';

	16#0000093C:
		F_EtherCAT_VendorIDtoString := 'Xi’an Aerospace Automation Co., Ltd';

	16#0000093D:
		F_EtherCAT_VendorIDtoString := 'Gal';

	16#0000093E:
		F_EtherCAT_VendorIDtoString := 'TOA Electronics Inc. Hamatou Company';

	16#00000940:
		F_EtherCAT_VendorIDtoString := 'Friedrich-Alexander-Universitat Erlangen-Nurnberg, Technische Fakultat';

	16#00000941:
		F_EtherCAT_VendorIDtoString := 'Sirius Electronic Systems s.r.l.';

	16#00000942:
		F_EtherCAT_VendorIDtoString := 'Chengdu InPlus Technology Co., Ltd.';

	16#00000943:
		F_EtherCAT_VendorIDtoString := 'MicroStep spol s.r.o.';

	16#00000944:
		F_EtherCAT_VendorIDtoString := 'Murata Machinery, Ltd.';

	16#00000946:
		F_EtherCAT_VendorIDtoString := 'Cabinplant A/S';

	16#00000948:
		F_EtherCAT_VendorIDtoString := 'Franka Robotics GmbH';

	16#0000094A:
		F_EtherCAT_VendorIDtoString := 'Smart Move GmbH';

	16#0000094B:
		F_EtherCAT_VendorIDtoString := 'Ampere Inc.';

	16#0000094C:
		F_EtherCAT_VendorIDtoString := 'Stichting Moving Bird (dba Project March)';

	16#0000094D:
		F_EtherCAT_VendorIDtoString := 'Imkon Endustriyel Otomasyon Sistemleri';

	16#0000094E:
		F_EtherCAT_VendorIDtoString := 'Tangshan Baichuan Intelligent Machine Co Ltd.';

	16#0000094F:
		F_EtherCAT_VendorIDtoString := 'Christian-Albrechts-Universitat zu Kiel';

	16#00000950:
		F_EtherCAT_VendorIDtoString := 'University of Lorraine, IUT Nancy-Brabois';

	16#00000951:
		F_EtherCAT_VendorIDtoString := 'Fraunhofer-Institut fur Optronik, Systemtechnik und Bildauswertung IOSB';

	16#00000952:
		F_EtherCAT_VendorIDtoString := 'IP-Automatika Kft.';

	16#00000953:
		F_EtherCAT_VendorIDtoString := 'EMKO Elektronik San. ve Tic. A.S.';

	16#00000954:
		F_EtherCAT_VendorIDtoString := 'FINE Inc.';

	16#00000955:
		F_EtherCAT_VendorIDtoString := 'Science and Technology Facilities Council, UK Astronomy Technology Centre (UK ATC)';

	16#00000956:
		F_EtherCAT_VendorIDtoString := 'ITmems s.r.l.';

	16#00000957:
		F_EtherCAT_VendorIDtoString := 'LumaSense Technologies, Inc.';

	16#00000958:
		F_EtherCAT_VendorIDtoString := 'ACUTRONIC Switzerland Ltd.';

	16#00000959:
		F_EtherCAT_VendorIDtoString := 'DieBie EngineeringTSC';

	16#0000095A:
		F_EtherCAT_VendorIDtoString := 'Procept Pty Ltd';

	16#0000095B:
		F_EtherCAT_VendorIDtoString := 'New Power Plasma Co., Ltd';

	16#0000095C:
		F_EtherCAT_VendorIDtoString := 'Advanced Mining Technology Center (AMTC)';

	16#0000095D:
		F_EtherCAT_VendorIDtoString := 'ASM Technology Singapore Pte Ltd.';

	16#0000095E:
		F_EtherCAT_VendorIDtoString := 'Weigl GmbH & Co KG';

	16#0000095F:
		F_EtherCAT_VendorIDtoString := 'Wagner International AG';

	16#00000960:
		F_EtherCAT_VendorIDtoString := 'Liebherr-Electronics and Drives GmbH';

	16#00000961:
		F_EtherCAT_VendorIDtoString := 'Mechatronics Labs S.r.l.';

	16#00000962:
		F_EtherCAT_VendorIDtoString := 'JIANGSU TORSUNG M&E CO.,LTD';

	16#00000963:
		F_EtherCAT_VendorIDtoString := 'Technicke služby BAHOZA s.r.o.';

	16#00000964:
		F_EtherCAT_VendorIDtoString := 'Siec Badawcza Lukasiewicz - Instytut Tele- i Radiotechniczny';

	16#00000965:
		F_EtherCAT_VendorIDtoString := 'Beijing Institute of Technology (BIT), School of Mechatronical Engineering';

	16#00000966:
		F_EtherCAT_VendorIDtoString := 'ElastiSense ApS';

	16#00000967:
		F_EtherCAT_VendorIDtoString := 'North China University of Technology, Beijing Key Laboratory of Fieldbus and Automation';

	16#00000968:
		F_EtherCAT_VendorIDtoString := 'Nidec Corporation';

	16#00000969:
		F_EtherCAT_VendorIDtoString := 'Hangzhou Zhishan Intelligent Control Technology Co. Ltd.';

	16#0000096A:
		F_EtherCAT_VendorIDtoString := 'Interface Devices Ltd.';

	16#0000096B:
		F_EtherCAT_VendorIDtoString := 'Nikon Corporation';

	16#0000096C:
		F_EtherCAT_VendorIDtoString := 'FCL COMPONENTS LIMITED';

	16#0000096D:
		F_EtherCAT_VendorIDtoString := 'Jiaxing Dealour Electric Technology Co.,Ltd.';

	16#0000096E:
		F_EtherCAT_VendorIDtoString := 'ETH Zurich, Department of Mechanical and Process Engineering (D-MAVT), Institute of Robotics and Intelligent Systems (IRIS)';

	16#0000096F:
		F_EtherCAT_VendorIDtoString := 'SURUGA Production Platform Co., Ltd.';

	16#00000970:
		F_EtherCAT_VendorIDtoString := 'Advanio Technology Co., Ltd.';

	16#00000971:
		F_EtherCAT_VendorIDtoString := 'EMBL Hamburg';

	16#00000972:
		F_EtherCAT_VendorIDtoString := 'Erle Robotics S.L.';

	16#00000973:
		F_EtherCAT_VendorIDtoString := 'SURUGA SEIKI CO., LTD.';

	16#00000974:
		F_EtherCAT_VendorIDtoString := 'EVA Robotics Pty Ltd';

	16#00000975:
		F_EtherCAT_VendorIDtoString := 'Beijing Etechwin Electric Co., Ltd.';

	16#00000976:
		F_EtherCAT_VendorIDtoString := 'KE Elektronik GmbH';

	16#00000977:
		F_EtherCAT_VendorIDtoString := 'ACCREA Bartlomiej Stanczyk';

	16#00000978:
		F_EtherCAT_VendorIDtoString := 'SCHUNK SE & Co. KG';

	16#00000979:
		F_EtherCAT_VendorIDtoString := 'Sciaky, Inc.';

	16#0000097A:
		F_EtherCAT_VendorIDtoString := 'Tokyo Robotics Inc.';

	16#0000097C:
		F_EtherCAT_VendorIDtoString := 'embeddeers GmbH';

	16#0000097D:
		F_EtherCAT_VendorIDtoString := 'GAMACO s.r.l.';

	16#0000097E:
		F_EtherCAT_VendorIDtoString := 'NPP VIUS, LLC';

	16#0000097F:
		F_EtherCAT_VendorIDtoString := 'ISG Industrielle Steuerungstechnik GmbH';

	16#00000980:
		F_EtherCAT_VendorIDtoString := 'FUJI ELECTRONICS CO.,LTD.';

	16#00000981:
		F_EtherCAT_VendorIDtoString := 'SHENZHEN MINGSU AUTOMATION EQUIPMENT CO., LTD';

	16#00000982:
		F_EtherCAT_VendorIDtoString := 'Jiangsu Ysphotech Technology Co.,LTD';

	16#00000983:
		F_EtherCAT_VendorIDtoString := 'Beijing JCZ Technology Co., Ltd.';

	16#00000984:
		F_EtherCAT_VendorIDtoString := 'DMG MORI CO., LTD.';

	16#00000985:
		F_EtherCAT_VendorIDtoString := 'TELSONIC AG';

	16#00000986:
		F_EtherCAT_VendorIDtoString := 'Tolomatic Inc.';

	16#00000987:
		F_EtherCAT_VendorIDtoString := 'NCWorks';

	16#00000988:
		F_EtherCAT_VendorIDtoString := 'Van Mierlo Ingenieursbureau BV';

	16#00000989:
		F_EtherCAT_VendorIDtoString := 'Control Technology Corporation';

	16#0000098A:
		F_EtherCAT_VendorIDtoString := 'TEAC Corporation';

	16#0000098D:
		F_EtherCAT_VendorIDtoString := 'Crossworks Inc.';

	16#0000098E:
		F_EtherCAT_VendorIDtoString := 'Agility Robotics';

	16#0000098F:
		F_EtherCAT_VendorIDtoString := 'ShenZhen Double CNC Tech Co., Ltd.';

	16#00000991:
		F_EtherCAT_VendorIDtoString := 'TSC Inc.';

	16#00000992:
		F_EtherCAT_VendorIDtoString := 'TE Connectivity Germany GmbH';

	16#00000993:
		F_EtherCAT_VendorIDtoString := 'Galli Brasil Comercio de Aparelhos Eletronicos Ltda.';

	16#00000994:
		F_EtherCAT_VendorIDtoString := 'Shenzhen YAKO Automation Technology Co.,Ltd';

	16#00000995:
		F_EtherCAT_VendorIDtoString := 'PRETTL Electronics India Pvt. Ltd.';

	16#00000997:
		F_EtherCAT_VendorIDtoString := 'Kehua Data Co., Ltd';

	16#00000998:
		F_EtherCAT_VendorIDtoString := 'Mayser GmbH & Co. KG';

	16#00000999:
		F_EtherCAT_VendorIDtoString := 'HAITIAN Plastics Machinery Group Co., Ltd';

	16#0000099A:
		F_EtherCAT_VendorIDtoString := 'Waco Giken Co., Ltd.';

	16#0000099B:
		F_EtherCAT_VendorIDtoString := 'Mike & Weingartner GmbH';

	16#0000099C:
		F_EtherCAT_VendorIDtoString := 'Ionicon Analytik Gesellschaft m.b.H.';

	16#0000099D:
		F_EtherCAT_VendorIDtoString := 'INESC TEC - Instituto de Engenharia de Sistemas e Computadores, Tecnologia e Ciencia';

	16#0000099E:
		F_EtherCAT_VendorIDtoString := '4automation';

	16#0000099F:
		F_EtherCAT_VendorIDtoString := 'Moog India Technology Center Pvt Ltd';

	16#000009A0:
		F_EtherCAT_VendorIDtoString := 'University of Cape Town, Department of Electrical Engineering';

	16#000009A1:
		F_EtherCAT_VendorIDtoString := 'Auris Health, Inc.';

	16#000009A2:
		F_EtherCAT_VendorIDtoString := 'Guangzhou Shiyuan Electronics Co., Ltd.';

	16#000009A3:
		F_EtherCAT_VendorIDtoString := 'Technische Universitat Ilmenau, Fakultat fur Maschinenbau, Fachgebiet Mechatronik';

	16#000009A4:
		F_EtherCAT_VendorIDtoString := 'HIT SPECIAL ROBOT CO.,LTD';

	16#000009A5:
		F_EtherCAT_VendorIDtoString := 'SmartDV Technologies India Private Limited';

	16#000009A6:
		F_EtherCAT_VendorIDtoString := 'Visitech AS';

	16#000009A7:
		F_EtherCAT_VendorIDtoString := 'Solartron Metrology Ltd.';

	16#000009A8:
		F_EtherCAT_VendorIDtoString := 'NKSystem K.K.';

	16#000009A9:
		F_EtherCAT_VendorIDtoString := 'INTRONIX spol. s.r.o.';

	16#000009AA:
		F_EtherCAT_VendorIDtoString := 'NetModule AG';

	16#000009AB:
		F_EtherCAT_VendorIDtoString := 'BZ Robot INC.';

	16#000009AC:
		F_EtherCAT_VendorIDtoString := 'PUES Corporation';

	16#000009AD:
		F_EtherCAT_VendorIDtoString := 'S.H.S. s.r.l.';

	16#000009AE:
		F_EtherCAT_VendorIDtoString := 'Manter International B.V.';

	16#000009AF:
		F_EtherCAT_VendorIDtoString := 'Delft University of Technology, Faculty of Aerospace Engineering';

	16#000009B0:
		F_EtherCAT_VendorIDtoString := 'GAMADE s.n.c. di Westfal Michele & C.';

	16#000009B1:
		F_EtherCAT_VendorIDtoString := 'ima-tec GmbH';

	16#000009B2:
		F_EtherCAT_VendorIDtoString := 'Evest Corporation';

	16#000009B3:
		F_EtherCAT_VendorIDtoString := 'SHINKO TECHNOS CO.,LTD.';

	16#000009B4:
		F_EtherCAT_VendorIDtoString := 'Sichuan University, School of Manufacturing Science and Engineering';

	16#000009B5:
		F_EtherCAT_VendorIDtoString := 'FLC Zbigniew Huber';

	16#000009B6:
		F_EtherCAT_VendorIDtoString := 'Taizhou Topcut-Bullmer Mechanical and Electrical Technology Co., Ltd.';

	16#000009B7:
		F_EtherCAT_VendorIDtoString := 'Shiratech Embedded Ltd.';

	16#000009B9:
		F_EtherCAT_VendorIDtoString := 'Eastern Logic Inc.';

	16#000009BA:
		F_EtherCAT_VendorIDtoString := 'WEBER Schraubautomaten GmbH';

	16#000009BB:
		F_EtherCAT_VendorIDtoString := 'Power Solution Network';

	16#000009BC:
		F_EtherCAT_VendorIDtoString := 'Advanced Thermal Sciences Corporation';

	16#000009BE:
		F_EtherCAT_VendorIDtoString := 'KITZ SCT Corporation';

	16#000009BF:
		F_EtherCAT_VendorIDtoString := 'Motorcon Inc.';

	16#000009C0:
		F_EtherCAT_VendorIDtoString := 'clownfish information technology GmbH';

	16#000009C1:
		F_EtherCAT_VendorIDtoString := 'RABE Engineering';

	16#000009C2:
		F_EtherCAT_VendorIDtoString := 'Ghost Robotics LLC';

	16#000009C3:
		F_EtherCAT_VendorIDtoString := 'Technische Universitat Graz';

	16#000009C5:
		F_EtherCAT_VendorIDtoString := 'Socionext Inc.';

	16#000009C6:
		F_EtherCAT_VendorIDtoString := 'Shenzhen Best Motion Technology Limited';

	16#000009C7:
		F_EtherCAT_VendorIDtoString := 'SPIE ESCAD Automation GmbH';

	16#000009C8:
		F_EtherCAT_VendorIDtoString := 'Universite Laval';

	16#000009CA:
		F_EtherCAT_VendorIDtoString := 'Akkodis Germany Consulting GmbH';

	16#000009CB:
		F_EtherCAT_VendorIDtoString := 'AMS - Gesellschaft fur Automatisierungs- und Me-Systemtechnik GmbH';

	16#000009CC:
		F_EtherCAT_VendorIDtoString := 'Techno-Holon Corporation';

	16#000009CD:
		F_EtherCAT_VendorIDtoString := 'J. Zimmer Maschinenbau GmbH';

	16#000009CE:
		F_EtherCAT_VendorIDtoString := 'e.sigma Technology GmbH';

	16#000009CF:
		F_EtherCAT_VendorIDtoString := 'OMRON AUTOMATION SYSTEM (HANGZHOU) CO.,LTD.';

	16#000009D0:
		F_EtherCAT_VendorIDtoString := 'Sof-Tek Integrators, Inc.';

	16#000009D1:
		F_EtherCAT_VendorIDtoString := 'CONTRINEX AG';

	16#000009D2:
		F_EtherCAT_VendorIDtoString := 'SISE SAS';

	16#000009D3:
		F_EtherCAT_VendorIDtoString := 'Christ Electronic Systems GmbH';

	16#000009D4:
		F_EtherCAT_VendorIDtoString := 'Nanjing LOYST Industrial Networks Co., Ltd.';

	16#000009D5:
		F_EtherCAT_VendorIDtoString := 'Spintrol Limited Corp.';

	16#000009D6:
		F_EtherCAT_VendorIDtoString := 'T.E.M.A. spa';

	16#000009D7:
		F_EtherCAT_VendorIDtoString := 'Ingenieurburo Fur IC-Technologie Franz Sprenger';

	16#000009D8:
		F_EtherCAT_VendorIDtoString := 'OPTO4L GmbH';

	16#000009D9:
		F_EtherCAT_VendorIDtoString := 'QuEST Global Services Pte. Ltd.';

	16#000009DB:
		F_EtherCAT_VendorIDtoString := 'ZIS Industrietechnik GmbH';

	16#000009DC:
		F_EtherCAT_VendorIDtoString := 'LOVATO Electric S.p.A';

	16#000009DD:
		F_EtherCAT_VendorIDtoString := 'E2M Technologies B.V.';

	16#000009DE:
		F_EtherCAT_VendorIDtoString := 'Zefatek Co., Ltd.';

	16#000009DF:
		F_EtherCAT_VendorIDtoString := 'Birket Engineering, Inc.';

	16#000009E0:
		F_EtherCAT_VendorIDtoString := 'JD Co., Ltd.';

	16#000009E1:
		F_EtherCAT_VendorIDtoString := 'Institut Clement Ader (ICA)';

	16#000009E2:
		F_EtherCAT_VendorIDtoString := 'OKANO CABLE CO., LTD';

	16#000009E3:
		F_EtherCAT_VendorIDtoString := 'Shenzhen OUR New Medical Technologies Development Co., Ltd.';

	16#000009E4:
		F_EtherCAT_VendorIDtoString := 'J. Schmalz GmbH';

	16#000009E5:
		F_EtherCAT_VendorIDtoString := 'Fives OTO S.p.a.';

	16#000009E6:
		F_EtherCAT_VendorIDtoString := 'INNOCONTACT CO.,LTD.';

	16#000009E7:
		F_EtherCAT_VendorIDtoString := 'silex technology, Inc.';

	16#000009E8:
		F_EtherCAT_VendorIDtoString := 'ShinMaywa Industries, LTD.';

	16#000009E9:
		F_EtherCAT_VendorIDtoString := 'ib prozessleittechnik GmbH & Co. KG';

	16#000009EA:
		F_EtherCAT_VendorIDtoString := 'EJTECH Inc.';

	16#000009EB:
		F_EtherCAT_VendorIDtoString := 'Shenzhen Hymson Laser Technologies Co.,Ltd.';

	16#000009EC:
		F_EtherCAT_VendorIDtoString := 'FlashCut CNC';

	16#000009ED:
		F_EtherCAT_VendorIDtoString := 'CTB Co., Ltd.';

	16#000009EE:
		F_EtherCAT_VendorIDtoString := 'Alexander Binzel Schweisstechnik GmbH & Co. KG';

	16#000009EF:
		F_EtherCAT_VendorIDtoString := 'SAWAMURA DENKI IND.CO.,LTD.';

	16#000009F0:
		F_EtherCAT_VendorIDtoString := 'Robowell Korea Co.';

	16#000009F1:
		F_EtherCAT_VendorIDtoString := 'MUSE Robotics Inc.';

	16#000009F2:
		F_EtherCAT_VendorIDtoString := 'Shenzhen WELLAUTO Technology CO., LTD.';

	16#000009F3:
		F_EtherCAT_VendorIDtoString := 'Primagest Inc.';

	16#000009F4:
		F_EtherCAT_VendorIDtoString := 'Aignep S.p.A.';

	16#000009F5:
		F_EtherCAT_VendorIDtoString := 'Pusan National University';

	16#000009F6:
		F_EtherCAT_VendorIDtoString := 'KUMOH MACH. & ELEC. CO., LTD.';

	16#000009F7:
		F_EtherCAT_VendorIDtoString := 'Chinese Academy of Sciences, Institute of Modern Physics (IMP)';

	16#000009F8:
		F_EtherCAT_VendorIDtoString := 'Houston Mechatronics, Inc.';

	16#000009F9:
		F_EtherCAT_VendorIDtoString := 'IAR Systems AB';

	16#000009FA:
		F_EtherCAT_VendorIDtoString := 'KOSHIDA KOREA CORPORATION';

	16#000009FB:
		F_EtherCAT_VendorIDtoString := 'Advanced Micro-Fabrication Equipment Inc.';

	16#000009FC:
		F_EtherCAT_VendorIDtoString := 'STEPHANIX S.A.';

	16#000009FD:
		F_EtherCAT_VendorIDtoString := 'CPI Technologies, Inc';

	16#000009FE:
		F_EtherCAT_VendorIDtoString := 'Harris Corporation';

	16#000009FF:
		F_EtherCAT_VendorIDtoString := 'Suzhou AGIOE Equipment Co. Ltd.';

	16#00000A00:
		F_EtherCAT_VendorIDtoString := 'OPTOELECTRONICS CO., LTD.';

	16#00000A01:
		F_EtherCAT_VendorIDtoString := 'Hitachi Energy Switzerland AG, Semiconductors';

	16#00000A02:
		F_EtherCAT_VendorIDtoString := 'FMS Force Measuring Systems AG';

	16#00000A03:
		F_EtherCAT_VendorIDtoString := 'Kulicke & Soffa Pte Ltd';

	16#00000A04:
		F_EtherCAT_VendorIDtoString := 'HEXMOTO Controls Pvt. Ltd';

	16#00000A05:
		F_EtherCAT_VendorIDtoString := 'Esautomotion s.r.l';

	16#00000A06:
		F_EtherCAT_VendorIDtoString := 'Canon ANELVA Corporation';

	16#00000A07:
		F_EtherCAT_VendorIDtoString := 'Glowbuzzer Ltd';

	16#00000A08:
		F_EtherCAT_VendorIDtoString := 'Technische Universitat Munchen, TUM School of Engineering and Design, Department of Mechanical Engineering, Lehrstuhl fur Angewandte Mechanik';

	16#00000A09:
		F_EtherCAT_VendorIDtoString := 'Beijing iTegva Technology Co., Ltd.';

	16#00000A0A:
		F_EtherCAT_VendorIDtoString := 'Zhejiang Wolong Servo Technology Co., Ltd.';

	16#00000A0B:
		F_EtherCAT_VendorIDtoString := 'SINOMACH Intelligence Technology Research Institute Co., Ltd.';

	16#00000A0C:
		F_EtherCAT_VendorIDtoString := 'Pusan National University, Department of Electronics Engineering, Embedded Control System Lab.';

	16#00000A0D:
		F_EtherCAT_VendorIDtoString := 'CRRC ZHUZHOU INSTITUTE CO.,LTD.';

	16#00000A0E:
		F_EtherCAT_VendorIDtoString := 'FATEK Automation Corporation';

	16#00000A0F:
		F_EtherCAT_VendorIDtoString := 'Racelogic Limited';

	16#00000A10:
		F_EtherCAT_VendorIDtoString := 'GRITEC AG';

	16#00000A11:
		F_EtherCAT_VendorIDtoString := 'Synhelion Germany GmbH';

	16#00000A12:
		F_EtherCAT_VendorIDtoString := 'National Technical University of Athens, School of Mechanical Engineering';

	16#00000A13:
		F_EtherCAT_VendorIDtoString := 'Changzhou GS Technology Co., Ltd.';

	16#00000A14:
		F_EtherCAT_VendorIDtoString := 'isel facility GmbH';

	16#00000A15:
		F_EtherCAT_VendorIDtoString := 'inotech Meter Calibration Systems GmbH';

	16#00000A16:
		F_EtherCAT_VendorIDtoString := 'HYUNDAI WIA CORP.';

	16#00000A17:
		F_EtherCAT_VendorIDtoString := 'DARPAMotion Ltd.';

	16#00000A18:
		F_EtherCAT_VendorIDtoString := 'MICRO TREND AUTOMATION CO.,LTD';

	16#00000A19:
		F_EtherCAT_VendorIDtoString := 'Suzhou Xiling Control Technology Co., Ltd.';

	16#00000A1A:
		F_EtherCAT_VendorIDtoString := 'UCAM Pvt. Ltd.';

	16#00000A1B:
		F_EtherCAT_VendorIDtoString := 'Thomas More Mechelen-Antwerpen vzw, Campus De Nayer, Department Technology & IT, EmSys Research Group';

	16#00000A1C:
		F_EtherCAT_VendorIDtoString := 'Planar Motor Incorporated';

	16#00000A1D:
		F_EtherCAT_VendorIDtoString := 'DYNAX Corporation';

	16#00000A1E:
		F_EtherCAT_VendorIDtoString := 'Mitsubishi Electric Corporation';

	16#00000A1F:
		F_EtherCAT_VendorIDtoString := 'Neways Technologies B.V.';

	16#00000A20:
		F_EtherCAT_VendorIDtoString := 'By Three projects Co.,Ltd.';

	16#00000A21:
		F_EtherCAT_VendorIDtoString := 'FMI Industrial Automation B.V.';

	16#00000A22:
		F_EtherCAT_VendorIDtoString := 'elecgator bvba';

	16#00000A23:
		F_EtherCAT_VendorIDtoString := 'EPA GmbH';

	16#00000A24:
		F_EtherCAT_VendorIDtoString := 'TESEC Corporation';

	16#00000A25:
		F_EtherCAT_VendorIDtoString := 'FUJITSU GENERAL ELECTRONICS LIMITED';

	16#00000A26:
		F_EtherCAT_VendorIDtoString := 'HOERBIGER Automatisierungstechnik GmbH';

	16#00000A27:
		F_EtherCAT_VendorIDtoString := 'RRRobotica Srl';

	16#00000A29:
		F_EtherCAT_VendorIDtoString := 'Servo Industrial Systems Co., Ltd.';

	16#00000A2A:
		F_EtherCAT_VendorIDtoString := 'Guangzhou Hongsen Servo Motor Co., Ltd.';

	16#00000A2C:
		F_EtherCAT_VendorIDtoString := 'U-System Co. Ltd.';

	16#00000A2D:
		F_EtherCAT_VendorIDtoString := 'Sarissa GmbH';

	16#00000A2E:
		F_EtherCAT_VendorIDtoString := 'Zitte Corporation';

	16#00000A2F:
		F_EtherCAT_VendorIDtoString := 'EOPTIS S.r.l.';

	16#00000A30:
		F_EtherCAT_VendorIDtoString := 'Aerotech, Inc.';

	16#00000A31:
		F_EtherCAT_VendorIDtoString := 'Cognizant Technology Solutions India Private Limited';

	16#00000A32:
		F_EtherCAT_VendorIDtoString := 'eSSys Co., Ltd.';

	16#00000A33:
		F_EtherCAT_VendorIDtoString := 'Alltec GmbH';

	16#00000A34:
		F_EtherCAT_VendorIDtoString := 'TDG Co.,Ltd.';

	16#00000A35:
		F_EtherCAT_VendorIDtoString := 'STAR SEIKI CO., LTD.';

	16#00000A36:
		F_EtherCAT_VendorIDtoString := 'SYNTEC TECHNOLOGY CO., LTD.';

	16#00000A38:
		F_EtherCAT_VendorIDtoString := 'COWIN.FA CO., Ltd.';

	16#00000A39:
		F_EtherCAT_VendorIDtoString := 'Rokae (Beijing) Robotics Technology Co.,Ltd.';

	16#00000A3A:
		F_EtherCAT_VendorIDtoString := 'JASA Packaging Systems BV';

	16#00000A3B:
		F_EtherCAT_VendorIDtoString := 'Tecnos G.A. Srl';

	16#00000A3C:
		F_EtherCAT_VendorIDtoString := 'NIPPON SYSTEMWARE CO.,LTD.';

	16#00000A3D:
		F_EtherCAT_VendorIDtoString := 'SPG Co., Ltd.';

	16#00000A3E:
		F_EtherCAT_VendorIDtoString := 'ISIT';

	16#00000A3F:
		F_EtherCAT_VendorIDtoString := 'Mirae Corporation';

	16#00000A40:
		F_EtherCAT_VendorIDtoString := 'STANLEY Engineered Fastening';

	16#00000A41:
		F_EtherCAT_VendorIDtoString := 'Beijing Does Robotics Co., Ltd.';

	16#00000A42:
		F_EtherCAT_VendorIDtoString := 'Amazipoint Technology Ltd.';

	16#00000A43:
		F_EtherCAT_VendorIDtoString := 'Arbite Robotics';

	16#00000A44:
		F_EtherCAT_VendorIDtoString := 'Lodz University of Technology, Faculty of Electrical, Electronic, Computer and Control Engineering';

	16#00000A45:
		F_EtherCAT_VendorIDtoString := 'Libertron Co., Ltd.';

	16#00000A46:
		F_EtherCAT_VendorIDtoString := 'FUJIFILM Healthcare Americas Corporation';

	16#00000A47:
		F_EtherCAT_VendorIDtoString := 'Kwangwoon University, College of Electronics and Information Engineering, School of Robotics';

	16#00000A48:
		F_EtherCAT_VendorIDtoString := 'SCANLAB GmbH';

	16#00000A49:
		F_EtherCAT_VendorIDtoString := 'Global Electronics Corporation';

	16#00000A4A:
		F_EtherCAT_VendorIDtoString := 'Embaix Consulting Dipl.-Ing Cord Elias';

	16#00000A4B:
		F_EtherCAT_VendorIDtoString := 'Wuxi Chihai Intelligent Technology Co., Ltd.';

	16#00000A4C:
		F_EtherCAT_VendorIDtoString := 'PAC TECH CO., LTD.';

	16#00000A4D:
		F_EtherCAT_VendorIDtoString := 'Tietech Co., Ltd.';

	16#00000A4E:
		F_EtherCAT_VendorIDtoString := 'Hauch & Bach ApS';

	16#00000A4F:
		F_EtherCAT_VendorIDtoString := 'OOO Vnedrencheskaya Firma Elna';

	16#00000A50:
		F_EtherCAT_VendorIDtoString := 'Shenzhen RuiDa Technology Co., Ltd.';

	16#00000A51:
		F_EtherCAT_VendorIDtoString := 'PTM mechatronics GmbH';

	16#00000A52:
		F_EtherCAT_VendorIDtoString := 'Schildknecht AG';

	16#00000A53:
		F_EtherCAT_VendorIDtoString := 'Shanghai Weihong Electronic Technology Co.,Ltd.';

	16#00000A54:
		F_EtherCAT_VendorIDtoString := 'OOO Compel';

	16#00000A55:
		F_EtherCAT_VendorIDtoString := 'Zixel sas di Beschin Augusto & C.';

	16#00000A57:
		F_EtherCAT_VendorIDtoString := 'Bender Robotics s.r.o.';

	16#00000A58:
		F_EtherCAT_VendorIDtoString := 'Power Standards Lab Inc.';

	16#00000A59:
		F_EtherCAT_VendorIDtoString := 'Ecole Polytechnique de Montreal, Electrical Engineering Department';

	16#00000A5A:
		F_EtherCAT_VendorIDtoString := 'Novanta IMS';

	16#00000A5B:
		F_EtherCAT_VendorIDtoString := 'Winservo (Xiamen) Electrical Technology Co., Ltd.';

	16#00000A5C:
		F_EtherCAT_VendorIDtoString := 'Weber Ultrasonics AG';

	16#00000A5D:
		F_EtherCAT_VendorIDtoString := 'NIDEC COPAL ELECTRONICS CORP.';

	16#00000A5E:
		F_EtherCAT_VendorIDtoString := 'Mattson Thermal Products GmbH';

	16#00000A5F:
		F_EtherCAT_VendorIDtoString := 'ReACT Technologies Inc.';

	16#00000A60:
		F_EtherCAT_VendorIDtoString := 'MILLAN Automation SAS';

	16#00000A61:
		F_EtherCAT_VendorIDtoString := 'ANDRITZ HYDRO GmbH';

	16#00000A62:
		F_EtherCAT_VendorIDtoString := 'Shenzhen Yuejiang Technology Co., Ltd.';

	16#00000A63:
		F_EtherCAT_VendorIDtoString := 'Fineline Limited';

	16#00000A64:
		F_EtherCAT_VendorIDtoString := 'OEMB SA';

	16#00000A65:
		F_EtherCAT_VendorIDtoString := 'Philoptics Co., Ltd.';

	16#00000A66:
		F_EtherCAT_VendorIDtoString := 'Vetaphone A/S';

	16#00000A67:
		F_EtherCAT_VendorIDtoString := 'Herkules-Resotec Elektronik GmbH';

	16#00000A68:
		F_EtherCAT_VendorIDtoString := 'ArtifactNoise, LLP';

	16#00000A69:
		F_EtherCAT_VendorIDtoString := 'DEPRAG SCHULZ GMBH u. CO. KG';

	16#00000A6A:
		F_EtherCAT_VendorIDtoString := 'Kinema AST S.r.l';

	16#00000A6B:
		F_EtherCAT_VendorIDtoString := 'ASAHI SURGICAL ROBOTICS CO.,LTD.';

	16#00000A6C:
		F_EtherCAT_VendorIDtoString := 'LLC "Plasmatic RnD"';

	16#00000A6D:
		F_EtherCAT_VendorIDtoString := 'Shanghai Tongyi Automation Technology Co., Ltd.';

	16#00000A6F:
		F_EtherCAT_VendorIDtoString := 'Plasmatreat GmbH';

	16#00000A70:
		F_EtherCAT_VendorIDtoString := 'Balt-System Ltd.';

	16#00000A71:
		F_EtherCAT_VendorIDtoString := 'Jack Sewing Machine Co., Ltd.';

	16#00000A72:
		F_EtherCAT_VendorIDtoString := 'Okura Yusoki Co., Ltd.';

	16#00000A73:
		F_EtherCAT_VendorIDtoString := 'CB7 Systems LLC';

	16#00000A74:
		F_EtherCAT_VendorIDtoString := 'Orotig S.r.l.';

	16#00000A75:
		F_EtherCAT_VendorIDtoString := 'SCHMIDT Technology GmbH';

	16#00000A76:
		F_EtherCAT_VendorIDtoString := 'Ingenieurburo Holtgrewe';

	16#00000A77:
		F_EtherCAT_VendorIDtoString := 'SWIGRO Additive Manufacturing Inc.';

	16#00000A78:
		F_EtherCAT_VendorIDtoString := 'SPI Developments Ltd.';

	16#00000A79:
		F_EtherCAT_VendorIDtoString := 'Shenzhen Xinchuan Electric Technology Co., Ltd.';

	16#00000A7A:
		F_EtherCAT_VendorIDtoString := 'Saab AB';

	16#00000A7B:
		F_EtherCAT_VendorIDtoString := 'Beckman Coulter K.K.';

	16#00000A7D:
		F_EtherCAT_VendorIDtoString := 'Crosscut Prototypes, LLC';

	16#00000A7E:
		F_EtherCAT_VendorIDtoString := 'Goertek Inc.';

	16#00000A7F:
		F_EtherCAT_VendorIDtoString := 'SHINKAWA LTD.';

	16#00000A80:
		F_EtherCAT_VendorIDtoString := 'adphos Innovative Technologies GmbH';

	16#00000A81:
		F_EtherCAT_VendorIDtoString := 'University of Stavanger, Faculty of Science and Technology';

	16#00000A82:
		F_EtherCAT_VendorIDtoString := 'RealSYS';

	16#00000A83:
		F_EtherCAT_VendorIDtoString := 'MTS Systems Corporation';

	16#00000A84:
		F_EtherCAT_VendorIDtoString := 'ZUKEN ELMIC, Inc.';

	16#00000A85:
		F_EtherCAT_VendorIDtoString := '"Power Supply Systems" Limited';

	16#00000A86:
		F_EtherCAT_VendorIDtoString := 'Nanjing Control Intelligent Technology Co.,Ltd.';

	16#00000A87:
		F_EtherCAT_VendorIDtoString := 'Laser Institute of Shandong Academy of Sciences';

	16#00000A88:
		F_EtherCAT_VendorIDtoString := 'Shenzhen Ruitech Mechanical and Electrical Technology Co.,Ltd.';

	16#00000A89:
		F_EtherCAT_VendorIDtoString := 'Shenzhen Hengyu Controller Technology Co., Ltd.';

	16#00000A8A:
		F_EtherCAT_VendorIDtoString := 'BE.services GmbH';

	16#00000A8B:
		F_EtherCAT_VendorIDtoString := 'Enertronica Santerno S.p.A.';

	16#00000A8C:
		F_EtherCAT_VendorIDtoString := 'O-DEAR INTERNATIONAL CORP.';

	16#00000A8D:
		F_EtherCAT_VendorIDtoString := 'Scanivalve Corp.';

	16#00000A8E:
		F_EtherCAT_VendorIDtoString := 'SMARTMOTION Co., Ltd.';

	16#00000A8F:
		F_EtherCAT_VendorIDtoString := 'TOYO SYSTEM Co., Ltd.';

	16#00000A90:
		F_EtherCAT_VendorIDtoString := 'Rheinmetall Electronics GmbH';

	16#00000A91:
		F_EtherCAT_VendorIDtoString := 'Vishay Nobel AB';

	16#00000A92:
		F_EtherCAT_VendorIDtoString := 'DMM Technology Corp.';

	16#00000A93:
		F_EtherCAT_VendorIDtoString := 'Crossmuller Pty Ltd';

	16#00000A94:
		F_EtherCAT_VendorIDtoString := 'ibg Prufcomputer GmbH';

	16#00000A95:
		F_EtherCAT_VendorIDtoString := 'NSK Ltd.';

	16#00000A96:
		F_EtherCAT_VendorIDtoString := 'ELEDUS s.r.o.';

	16#00000A97:
		F_EtherCAT_VendorIDtoString := 'Baldwin Technology GmbH';

	16#00000A98:
		F_EtherCAT_VendorIDtoString := 'Blum-Novotest GmbH';

	16#00000A99:
		F_EtherCAT_VendorIDtoString := 'KROHNE Messtechnik GmbH';

	16#00000A9B:
		F_EtherCAT_VendorIDtoString := 'Shenzhen ECON Technology Co.,Ltd.';

	16#00000A9C:
		F_EtherCAT_VendorIDtoString := 'National Institute of Advanced Industrial Science and Technology (AIST), Intelligent Systems Research Institute (ISRI)';

	16#00000A9E:
		F_EtherCAT_VendorIDtoString := 'ZELTWANGER Leaktesting & Automation GmbH';

	16#00000A9F:
		F_EtherCAT_VendorIDtoString := 'CoSynth GmbH & Co. KG';

	16#00000AA0:
		F_EtherCAT_VendorIDtoString := 'Technical Development Corporation';

	16#00000AA1:
		F_EtherCAT_VendorIDtoString := 'AREVO INC.';

	16#00000AA2:
		F_EtherCAT_VendorIDtoString := 'MTT Corporation';

	16#00000AA3:
		F_EtherCAT_VendorIDtoString := 'MIS Corporation';

	16#00000AA4:
		F_EtherCAT_VendorIDtoString := 'Mackware GmbH';

	16#00000AA5:
		F_EtherCAT_VendorIDtoString := 'Reno Sub-Systems Inc.';

	16#00000AA6:
		F_EtherCAT_VendorIDtoString := 'BARBERAN S.A.';

	16#00000AA7:
		F_EtherCAT_VendorIDtoString := 'Stratasys, Inc.';

	16#00000AA8:
		F_EtherCAT_VendorIDtoString := 'DEPUSH Technology Co.,Ltd.';

	16#00000AA9:
		F_EtherCAT_VendorIDtoString := 'Justus-Liebig-Universitat Gieen, I. Physikalisches Institut, Arbeitsgruppe Atom- und Molekulphysik';

	16#00000AAA:
		F_EtherCAT_VendorIDtoString := 'Think Surgical, Inc.';

	16#00000AAB:
		F_EtherCAT_VendorIDtoString := 'Zhengzhou Runhua Intelligent Equipment Co., Ltd.';

	16#00000AAC:
		F_EtherCAT_VendorIDtoString := 'Unipulse Corporation';

	16#00000AAD:
		F_EtherCAT_VendorIDtoString := 'Foshan City Coyo Precision Machinery Manufacturing Co. Ltd';

	16#00000AAE:
		F_EtherCAT_VendorIDtoString := 'Teknix Argentina SRL';

	16#00000AAF:
		F_EtherCAT_VendorIDtoString := 'TDK Corporation';

	16#00000AB0:
		F_EtherCAT_VendorIDtoString := 'HYUNDAI MOVEX';

	16#00000AB1:
		F_EtherCAT_VendorIDtoString := 'The Charles Stark Draper Laboratory, Inc.';

	16#00000AB2:
		F_EtherCAT_VendorIDtoString := 'Technische Universitat Berlin, Fakultat Elektrotechnik und Informatik, Fachgebiet Telekommunikationsnetze';

	16#00000AB3:
		F_EtherCAT_VendorIDtoString := 'Star Asia Trading Pte. Ltd.';

	16#00000AB4:
		F_EtherCAT_VendorIDtoString := 'Jiangsu Fulling Motor Technology Co., Ltd.';

	16#00000AB5:
		F_EtherCAT_VendorIDtoString := 'Shenzhen Qinglan Automation Technology Co.,Ltd';

	16#00000AB6:
		F_EtherCAT_VendorIDtoString := 'Beijing Hollysys Electric Technology Co., Ltd.';

	16#00000AB7:
		F_EtherCAT_VendorIDtoString := 'ANTRIMON Group AG';

	16#00000AB8:
		F_EtherCAT_VendorIDtoString := 'Technische Universitat Dresden, Fakultat Maschinenwesen, Institut fur Mechatronischen Maschinenbau, Professur fur Werkzeugmaschinenentwicklung und adaptive Steuerungen';

	16#00000AB9:
		F_EtherCAT_VendorIDtoString := 'MikroElektronika d.o.o.';

	16#00000ABA:
		F_EtherCAT_VendorIDtoString := 'Sasken Technologies Limited';

	16#00000ABB:
		F_EtherCAT_VendorIDtoString := 'ABB AS Corporate Research';

	16#00000ABD:
		F_EtherCAT_VendorIDtoString := 'STIGAL';

	16#00000ABE:
		F_EtherCAT_VendorIDtoString := 'TnS Co., Ltd';

	16#00000ABF:
		F_EtherCAT_VendorIDtoString := 'PAIX Co.,Ltd';

	16#00000AC0:
		F_EtherCAT_VendorIDtoString := 'Senfit Ltd.';

	16#00000AC1:
		F_EtherCAT_VendorIDtoString := 'Promaster Technology Corporation';

	16#00000AC2:
		F_EtherCAT_VendorIDtoString := 'CRSC Urban Rail Transit Technology Co.,Ltd';

	16#00000AC3:
		F_EtherCAT_VendorIDtoString := 'Anthony Best Dynamics Ltd.';

	16#00000AC4:
		F_EtherCAT_VendorIDtoString := 'TVM Signalling and Transportation Systems Pvt. Ltd';

	16#00000AC5:
		F_EtherCAT_VendorIDtoString := 'neuroConn GmbH';

	16#00000AC6:
		F_EtherCAT_VendorIDtoString := 'Servelec Technologies Pty Ltd';

	16#00000AC7:
		F_EtherCAT_VendorIDtoString := 'Stereotaxis, Inc.';

	16#00000AC8:
		F_EtherCAT_VendorIDtoString := 'National Formosa University, College of Engineering';

	16#00000AC9:
		F_EtherCAT_VendorIDtoString := 'Alma Mater Studiorum - Universita di Bologna, Department of Electrical, Electronic and Information Engineering “Guglielmo Marconi”, Laboratory of Automation and Robotics';

	16#00000ACA:
		F_EtherCAT_VendorIDtoString := 'Centroid Corporation';

	16#00000ACC:
		F_EtherCAT_VendorIDtoString := 'Nidec Motor Corporation';

	16#00000ACD:
		F_EtherCAT_VendorIDtoString := 'NAVER LABS Corp.';

	16#00000ACE:
		F_EtherCAT_VendorIDtoString := 'Hitachi Industry & Control Solutions, Ltd.';

	16#00000ACF:
		F_EtherCAT_VendorIDtoString := 'Thermo Fisher Scientific Messtechnik GmbH';

	16#00000AD0:
		F_EtherCAT_VendorIDtoString := 'JSC "T-Platforms"';

	16#00000AD1:
		F_EtherCAT_VendorIDtoString := 'Halodi Robotics AS';

	16#00000AD2:
		F_EtherCAT_VendorIDtoString := 'Skala Sp. z o.o.';

	16#00000AD3:
		F_EtherCAT_VendorIDtoString := 'Jin Solution Co., Ltd.';

	16#00000AD4:
		F_EtherCAT_VendorIDtoString := 'KingSemi Co.,Ltd';

